StepDone := ExecuteSkill.Done;
END_ACTION

ACTION Transport1_active:
StepDone := FALSE;

//Skill auswählen
ExecuteSkill.SkillID 		:= 1320;
ExecuteSkill.SkillName	 	:= 'Name';

//Parameter setzen

ExecuteSkill.Parameter[3].ID := 3;
ExecuteSkill.Parameter[3].Name := 'Velocity';
ExecuteSkill.Parameter[3].Value := 2500;



ExecuteSkill.Parameter[4].ID := 4 ;
ExecuteSkill.Parameter[4].Name := 'Acceleration';
ExecuteSkill.Parameter[4].Value := 1000 ;



ExecuteSkill.Parameter[1].ID := 1;
ExecuteSkill.Parameter[1].Name := 'TargetPosition X';
ExecuteSkill.Parameter[1].Value := 3200 ;
ExecuteSkill.Parameter[1].StringValue := '#DP#2#XPosition' ;




ExecuteSkill.Parameter[2].ID := 2;
ExecuteSkill.Parameter[2].Name := 'TargetPosition Z';
ExecuteSkill.Parameter[2].Value := ZCookieModule;


(*
ExecuteSkill.Parameter[5].ID := ;
ExecuteSkill.Parameter[5].Name := '';
ExecuteSkill.Parameter[5].Value := ;
*)



ExecuteSkill();

StepDone := ExecuteSkill.Done;
END_ACTION

ACTION BlockBeiTopping_active:
StepDone := FALSE;

//Skill auswählen
ExecuteSkill.SkillID 		:= 1315;
ExecuteSkill.SkillName	 	:= 'Block';

//Parameter setzen

ExecuteSkill.Parameter[1].ID := 1;
ExecuteSkill.Parameter[1].Name := 'TaskID';
ExecuteSkill.Parameter[1].Value := 130;


(*
ExecuteSkill.Parameter[2].ID := ;
ExecuteSkill.Parameter[2].Name := '';
ExecuteSkill.Parameter[2].Value := ;
*)

(*
ExecuteSkill.Parameter[3].ID := ;
ExecuteSkill.Parameter[3].Name := '';
ExecuteSkill.Parameter[3].Value := ;
*)

(*
ExecuteSkill.Parameter[4].ID := ;
ExecuteSkill.Parameter[4].Name := '';
ExecuteSkill.Parameter[4].Value := ;
*)

(*
ExecuteSkill.Parameter[5].ID := ;
ExecuteSkill.Parameter[5].Name := '';
ExecuteSkill.Parameter[5].Value := ;
*)



ExecuteSkill();

StepDone := ExecuteSkill.Done;
END_ACTION

ACTION Topping_active:
StepDone := FALSE;

//Skill auswählen
ExecuteSkill.SkillID 		:= 1210;
ExecuteSkill.SkillName	 	:= 'Topping';

//Parameter setzen
(*
ExecuteSkill.Parameter[1].ID := 1;
ExecuteSkill.Parameter[1].Name := 'TaskID';
ExecuteSkill.Parameter[1].Value := 130;
*)
(*
ExecuteSkill.Parameter[2].ID := ;
ExecuteSkill.Parameter[2].Name := '';
ExecuteSkill.Parameter[2].Value := ;
*)

(*
ExecuteSkill.Parameter[3].ID := ;
ExecuteSkill.Parameter[3].Name := '';
ExecuteSkill.Parameter[3].Value := ;
*)

(*
ExecuteSkill.Parameter[4].ID := ;
ExecuteSkill.Parameter[4].Name := '';
ExecuteSkill.Parameter[4].Value := ;
*)

(*
ExecuteSkill.Parameter[5].ID := ;
ExecuteSkill.Parameter[5].Name := '';
ExecuteSkill.Parameter[5].Value := ;
*)

ExecuteSkill();

StepDone := ExecuteSkill.Done;
END_ACTION

ACTION TransportToTopping_active:
StepDone := FALSE;

//Skill auswählen
ExecuteSkill.SkillID 		:= 1320;
ExecuteSkill.SkillName	 	:= 'Transport';

//Parameter setzen

ExecuteSkill.Parameter[3].ID := 3;
ExecuteSkill.Parameter[3].Name := 'Velocity';
ExecuteSkill.Parameter[3].Value := 1500;



ExecuteSkill.Parameter[1].ID :=  1;
ExecuteSkill.Parameter[1].Name := 'TargetPosition X';
ExecuteSkill.Parameter[1].Value := 30 ;
ExecuteSkill.Parameter[1].StringValue := '#DP#2#XPosition';



ExecuteSkill.Parameter[2].ID := 2;
ExecuteSkill.Parameter[2].Name := 'TargetPosition Z';
ExecuteSkill.Parameter[2].Value := ZCremeModule ;

ExecuteSkill();

StepDone := ExecuteSkill.Done;
END_ACTION

ACTION MODULESkill_active:
StepDone := FALSE;
RecipeDone := FALSE;
//Skill auswählen
ExecuteSkill.SkillID 		:= 1010;
ExecuteSkill.SkillName	 	:= 'Cookie ausgeben';





ExecuteSkill();

StepDone := ExecuteSkill.Done;
END_ACTION

ACTION Unblock1_active:
StepDone := FALSE;

//Skill auswählen
ExecuteSkill.SkillID 		:= 1316;
ExecuteSkill.SkillName	 	:= 'Unblock';

//Parameter setzen

ExecuteSkill.Parameter[1].ID := 1;
ExecuteSkill.Parameter[1].Name := 'TaskID';
ExecuteSkill.Parameter[1].Value := 128 ;


(*
ExecuteSkill.Parameter[2].ID := ;
ExecuteSkill.Parameter[2].Name := '';
ExecuteSkill.Parameter[2].Value := ;
*)

(*
ExecuteSkill.Parameter[3].ID := ;
ExecuteSkill.Parameter[3].Name := '';
ExecuteSkill.Parameter[3].Value := ;
*)

(*
ExecuteSkill.Parameter[4].ID := ;
ExecuteSkill.Parameter[4].Name := '';
ExecuteSkill.Parameter[4].Value := ;
*)

(*
ExecuteSkill.Parameter[5].ID := ;
ExecuteSkill.Parameter[5].Name := '';
ExecuteSkill.Parameter[5].Value := ;
*)



ExecuteSkill();

StepDone := ExecuteSkill.Done;
END_ACTION

ACTION Block1_active:
StepDone := FALSE;

//Skill auswählen
ExecuteSkill.SkillID 		:= 1315;
ExecuteSkill.SkillName	 	:= 'Block';

//Parameter setzen

ExecuteSkill.Parameter[1].ID := 1;
ExecuteSkill.Parameter[1].Name := 'TaskID';
ExecuteSkill.Parameter[1].Value := 127;


(*
ExecuteSkill.Parameter[2].ID := ;
ExecuteSkill.Parameter[2].Name := '';
ExecuteSkill.Parameter[2].Value := ;
*)

(*
ExecuteSkill.Parameter[3].ID := ;
ExecuteSkill.Parameter[3].Name := '';
ExecuteSkill.Parameter[3].Value := ;
*)

(*
ExecuteSkill.Parameter[4].ID := ;
ExecuteSkill.Parameter[4].Name := '';
ExecuteSkill.Parameter[4].Value := ;
*)

(*
ExecuteSkill.Parameter[5].ID := ;
ExecuteSkill.Parameter[5].Name := '';
ExecuteSkill.Parameter[5].Value := ;
*)



ExecuteSkill();

StepDone := ExecuteSkill.Done;
END_ACTION

ACTION Transport_active:
StepDone := FALSE;

//Skill auswählen
ExecuteSkill.SkillID 		:= 1320;
ExecuteSkill.SkillName	 	:= 'Transport';

//Parameter setzen

ExecuteSkill.Parameter[3].ID :=3 ;
ExecuteSkill.Parameter[3].Name := 'Velocity';
ExecuteSkill.Parameter[3].Value := 1500;



ExecuteSkill.Parameter[1].ID :=1 ;
ExecuteSkill.Parameter[1].Name := 'TargetPosition X';
ExecuteSkill.Parameter[1].StringValue := '#DP#2#XPosition';
ExecuteSkill.Parameter[1].Value := 200 ;


ExecuteSkill.Parameter[2].ID := 2 ;
ExecuteSkill.Parameter[2].Name := 'TargetPosition Z';
ExecuteSkill.Parameter[2].Value := 90 ;



ExecuteSkill.Parameter[4].ID := 4 ;
ExecuteSkill.Parameter[4].Name := 'Acceleration';
ExecuteSkill.Parameter[4].Value := 4500;


(*
ExecuteSkill.Parameter[5].ID := ;
ExecuteSkill.Parameter[5].Name := '';
ExecuteSkill.Parameter[5].Value := ;
*)



ExecuteSkill();

StepDone := ExecuteSkill.Done;
END_ACTION

ACTION Block2_active:
StepDone := FALSE;

//Skill auswählen
ExecuteSkill.SkillID 		:= 1315;
ExecuteSkill.SkillName	 	:= 'Block';

//Parameter setzen

ExecuteSkill.Parameter[1].ID := 1;
ExecuteSkill.Parameter[1].Name := 'TaskID';
ExecuteSkill.Parameter[1].Value := 130;


(*
ExecuteSkill.Parameter[2].ID := ;
ExecuteSkill.Parameter[2].Name := '';
ExecuteSkill.Parameter[2].Value := ;
*)

(*
ExecuteSkill.Parameter[3].ID := ;
ExecuteSkill.Parameter[3].Name := '';
ExecuteSkill.Parameter[3].Value := ;
*)

(*
ExecuteSkill.Parameter[4].ID := ;
ExecuteSkill.Parameter[4].Name := '';
ExecuteSkill.Parameter[4].Value := ;
*)

(*
ExecuteSkill.Parameter[5].ID := ;
ExecuteSkill.Parameter[5].Name := '';
ExecuteSkill.Parameter[5].Value := ;
*)



ExecuteSkill();

StepDone := ExecuteSkill.Done;
END_ACTION

ACTION Block_active:
StepDone := FALSE;

//Skill auswählen
ExecuteSkill.SkillID 		:= 1315;
ExecuteSkill.SkillName	 	:= 'Block';

//Parameter setzen

ExecuteSkill.Parameter[1].ID := 1;
ExecuteSkill.Parameter[1].Name := 'TaskID';
ExecuteSkill.Parameter[1].Value := 124;


(*
ExecuteSkill.Parameter[2].ID := ;
ExecuteSkill.Parameter[2].Name := '';
ExecuteSkill.Parameter[2].Value := ;
*)

(*
ExecuteSkill.Parameter[3].ID := ;
ExecuteSkill.Parameter[3].Name := '';
ExecuteSkill.Parameter[3].Value := ;
*)

(*
ExecuteSkill.Parameter[4].ID := ;
ExecuteSkill.Parameter[4].Name := '';
ExecuteSkill.Parameter[4].Value := ;
*)

(*
ExecuteSkill.Parameter[5].ID := ;
ExecuteSkill.Parameter[5].Name := '';
ExecuteSkill.Parameter[5].Value := ;
*)



ExecuteSkill();

StepDone := ExecuteSkill.Done;
END_ACTION

ACTION Reserve_active:
StepDone := FALSE;
RecipeDone := FALSE;
//Skill auswählen
ExecuteSkill.SkillID 		:= 1310;
ExecuteSkill.SkillName	 	:= 'Reserve';

//Parameter setzen

ExecuteSkill.Parameter[1].ID := 1;
ExecuteSkill.Parameter[1].Name := 'TaskID';
ExecuteSkill.Parameter[1].Value := 123;


(*
ExecuteSkill.Parameter[2].ID := ;
ExecuteSkill.Parameter[2].Name := '';
ExecuteSkill.Parameter[2].Value := ;
*)

(*
ExecuteSkill.Parameter[3].ID := ;
ExecuteSkill.Parameter[3].Name := '';
ExecuteSkill.Parameter[3].Value := ;
*)

(*
ExecuteSkill.Parameter[4].ID := ;
ExecuteSkill.Parameter[4].Name := '';
ExecuteSkill.Parameter[4].Value := ;
*)

(*
ExecuteSkill.Parameter[5].ID := ;
ExecuteSkill.Parameter[5].Name := '';
ExecuteSkill.Parameter[5].Value := ;
*)



ExecuteSkill();

StepDone := ExecuteSkill.Done;
END_ACTION

ACTION Production0_active:
StepDone := FALSE;
RecipeDone := FALSE;
//Skill auswählen
ExecuteSkill.SkillID 		:= 1337;
ExecuteSkill.SkillName	 	:= 'Testmodul1';

ExecuteSkill();

StepDone := ExecuteSkill.Done;
END_ACTION

END_FUNCTION_BLOCK

// ---- POUs/Recipes/Recipe_10054_FreePassion_special.TcPOU
FUNCTION_BLOCK Recipe_10054_FreePassion_special
VAR_INPUT
	execute: BOOL;
	Order: DUT_RECIPEORDER;
END_VAR
VAR_OUTPUT
	RecipeInfo: DUT_RECIPEOFFER;
	RecipeDone: BOOL;
	InitDone: BOOL;
END_VAR
VAR
	userparametersum: LREAL;
	StepDone: BOOL;
	i: INT;
END_VAR

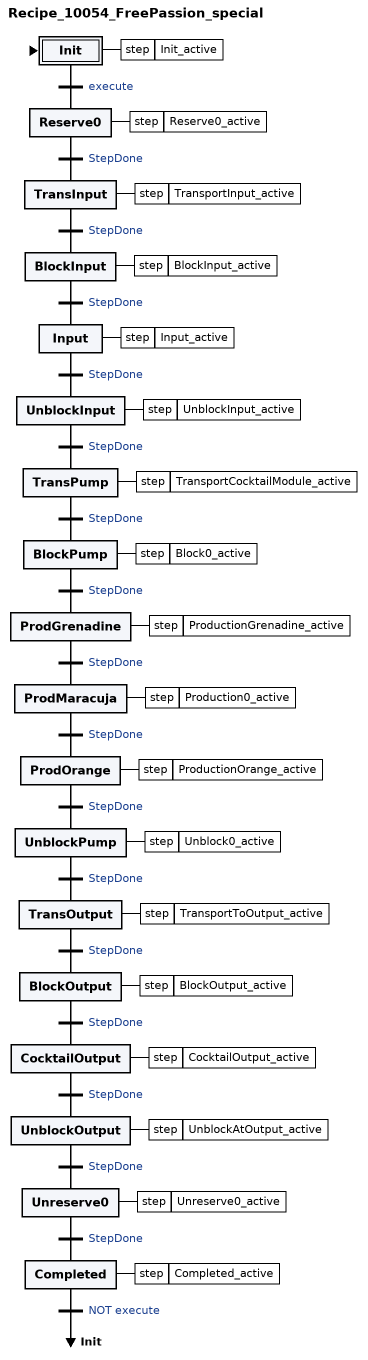
INITIAL_STEP Init:
    Init_active(N);  // step action
END_STEP
TRANSITION FROM Init TO Reserve0
    := execute;
END_TRANSITION
STEP Reserve0:
    Reserve0_active(N);  // step action
END_STEP
TRANSITION FROM Reserve0 TO TransInput
    := StepDone;
END_TRANSITION
STEP TransInput:
    TransportInput_active(N);  // step action
END_STEP
TRANSITION FROM TransInput TO BlockInput
    := StepDone;
END_TRANSITION
STEP BlockInput:
    BlockInput_active(N);  // step action
END_STEP
TRANSITION FROM BlockInput TO Input
    := StepDone;
END_TRANSITION
STEP Input:
    Input_active(N);  // step action
END_STEP
TRANSITION FROM Input TO UnblockInput
    := StepDone;
END_TRANSITION
STEP UnblockInput:
    UnblockInput_active(N);  // step action
END_STEP
TRANSITION FROM UnblockInput TO TransPump
    := StepDone;
END_TRANSITION
STEP TransPump:
    TransportCocktailModule_active(N);  // step action
END_STEP
TRANSITION FROM TransPump TO BlockPump
    := StepDone;
END_TRANSITION
STEP BlockPump:
    Block0_active(N);  // step action
END_STEP
TRANSITION FROM BlockPump TO ProdGrenadine
    := StepDone;
END_TRANSITION
STEP ProdGrenadine:
    ProductionGrenadine_active(N);  // step action
END_STEP
TRANSITION FROM ProdGrenadine TO ProdMaracuja
    := StepDone;
END_TRANSITION
STEP ProdMaracuja:
    Production0_active(N);  // step action
END_STEP
TRANSITION FROM ProdMaracuja TO ProdOrange
    := StepDone;
END_TRANSITION
STEP ProdOrange:
    ProductionOrange_active(N);  // step action
END_STEP
TRANSITION FROM ProdOrange TO UnblockPump
    := StepDone;
END_TRANSITION
STEP UnblockPump:
    Unblock0_active(N);  // step action
END_STEP
TRANSITION FROM UnblockPump TO TransOutput
    := StepDone;
END_TRANSITION
STEP TransOutput:
    TransportToOutput_active(N);  // step action
END_STEP
TRANSITION FROM TransOutput TO BlockOutput
    := StepDone;
END_TRANSITION
STEP BlockOutput:
    BlockOutput_active(N);  // step action
END_STEP
TRANSITION FROM BlockOutput TO CocktailOutput
    := StepDone;
END_TRANSITION
STEP CocktailOutput:
    CocktailOutput_active(N);  // step action
END_STEP
TRANSITION FROM CocktailOutput TO UnblockOutput
    := StepDone;
END_TRANSITION
STEP UnblockOutput:
    UnblockAtOutput_active(N);  // step action
END_STEP
TRANSITION FROM UnblockOutput TO Unreserve0
    := StepDone;
END_TRANSITION
STEP Unreserve0:
    Unreserve0_active(N);  // step action
END_STEP
TRANSITION FROM Unreserve0 TO Completed
    := StepDone;
END_TRANSITION
STEP Completed:
    Completed_active(N);  // step action
END_STEP
TRANSITION FROM Completed TO Init
    := NOT execute;
END_TRANSITION

ACTION Production0_active:
StepDone := FALSE;

userparametersum := 0;
FOR i := 1 TO UserParameterCnt DO
	IF NOT (order.UserParameter[i].Value = 0) THEN
		userparametersum := userparametersum + order.UserParameter[i].Value;
	
	END_IF
END_FOR
IF userparametersum = 0 THEN
userparametersum := -1;
END_IF
//Skill auswählen
ExecuteSkill.SkillID 		:= 1113;
ExecuteSkill.SkillName	 	:= 'Marajuca Juice';

//Parameter setzen

ExecuteSkill.Parameter[0].ID := 1;
ExecuteSkill.Parameter[0].Name := 'Quantity';
//order.userParameter[0] = amount
ExecuteSkill.Parameter[0].Value := order.UserParameter[0].Value * order.UserParameter[1].Value / userparametersum;//Summe aller Zutatenmengen;


(*
ExecuteSkill.Parameter[2].ID := ;
ExecuteSkill.Parameter[2].Name := '';
ExecuteSkill.Parameter[2].Value := ;
*)

(*
ExecuteSkill.Parameter[3].ID := ;
ExecuteSkill.Parameter[3].Name := '';
ExecuteSkill.Parameter[3].Value := ;
*)

(*
ExecuteSkill.Parameter[4].ID := ;
ExecuteSkill.Parameter[4].Name := '';
ExecuteSkill.Parameter[4].Value := ;
*)

(*
ExecuteSkill.Parameter[5].ID := ;
ExecuteSkill.Parameter[5].Name := '';
ExecuteSkill.Parameter[5].Value := ;
*)



ExecuteSkill();

StepDone := ExecuteSkill.Done;
END_ACTION

ACTION TransportInput_active:
StepDone := FALSE;

//Skill auswählen
ExecuteSkill.SkillID 		:= 1320;
ExecuteSkill.SkillName	 	:= 'Transport';

//Parameter setzen

ExecuteSkill.Parameter[3].ID := 3;
ExecuteSkill.Parameter[3].Name := 'Velocity';
ExecuteSkill.Parameter[3].Value := 1500;



ExecuteSkill.Parameter[1].ID :=  1;
ExecuteSkill.Parameter[1].Name := 'TargetPosition X';
ExecuteSkill.Parameter[1].Value := 30 ;
ExecuteSkill.Parameter[1].StringValue := '#DP#2#XPosition';



ExecuteSkill.Parameter[2].ID := 2;
ExecuteSkill.Parameter[2].Name := 'TargetPosition Z';
ExecuteSkill.Parameter[2].Value := 100;// ZCookieModule - ZCookieModuleCalibration - 2* Cookiethickness + toppingthickness+ Preasureheight  ;



(*
ExecuteSkill.Parameter[4].ID := 4;
ExecuteSkill.Parameter[4].Name := 'Acceleration';
ExecuteSkill.Parameter[4].Value := 0 ;
*)

(*
ExecuteSkill.Parameter[5].ID := ;
ExecuteSkill.Parameter[5].Name := '';
ExecuteSkill.Parameter[5].Value := ;
*)



ExecuteSkill();

StepDone := ExecuteSkill.Done;
END_ACTION

ACTION BlockOutput_active:
StepDone := FALSE;

//Skill auswählen
ExecuteSkill.SkillID 		:= 1315;
ExecuteSkill.SkillName	 	:= 'Block';

//Parameter setzen

ExecuteSkill.Parameter[1].ID := 1;
ExecuteSkill.Parameter[1].Name := 'TaskID';
ExecuteSkill.Parameter[1].Value := Order.TaskID;


(*
ExecuteSkill.Parameter[2].ID := ;
ExecuteSkill.Parameter[2].Name := '';
ExecuteSkill.Parameter[2].Value := ;
*)

(*
ExecuteSkill.Parameter[3].ID := ;
ExecuteSkill.Parameter[3].Name := '';
ExecuteSkill.Parameter[3].Value := ;
*)

(*
ExecuteSkill.Parameter[4].ID := ;
ExecuteSkill.Parameter[4].Name := '';
ExecuteSkill.Parameter[4].Value := ;
*)

(*
ExecuteSkill.Parameter[5].ID := ;
ExecuteSkill.Parameter[5].Name := '';
ExecuteSkill.Parameter[5].Value := ;
*)



ExecuteSkill();

StepDone := ExecuteSkill.Done;
END_ACTION

ACTION ProductionGrenadine_active:
StepDone := FALSE;

//Skill auswählen
ExecuteSkill.SkillID 		:= 1121;
ExecuteSkill.SkillName	 	:= 'Batida de Coco';

//Parameter setzen

ExecuteSkill.Parameter[0].ID := 1;
ExecuteSkill.Parameter[0].Name := 'Quantity';
//order.userParameter[0] = amount
ExecuteSkill.Parameter[0].Value := order.UserParameter[0].Value * order.UserParameter[3].Value / userparametersum; //Summe aller Zutatenmengen;



(*
ExecuteSkill.Parameter[2].ID := ;
ExecuteSkill.Parameter[2].Name := '';
ExecuteSkill.Parameter[2].Value := ;
*)

(*
ExecuteSkill.Parameter[3].ID := ;
ExecuteSkill.Parameter[3].Name := '';
ExecuteSkill.Parameter[3].Value := ;
*)

(*
ExecuteSkill.Parameter[4].ID := ;
ExecuteSkill.Parameter[4].Name := '';
ExecuteSkill.Parameter[4].Value := ;
*)

(*
ExecuteSkill.Parameter[5].ID := ;
ExecuteSkill.Parameter[5].Name := '';
ExecuteSkill.Parameter[5].Value := ;
*)



ExecuteSkill();

StepDone := ExecuteSkill.Done;
END_ACTION

ACTION Unreserve0_active:
StepDone := FALSE;

//Skill auswählen
ExecuteSkill.SkillID 		:= 1311;
ExecuteSkill.SkillName	 	:= 'Unreserve';

//Parameter setzen

ExecuteSkill.Parameter[1].ID := 1;
ExecuteSkill.Parameter[1].Name := 'TaskID';
ExecuteSkill.Parameter[1].Value := Order.TaskID;


(*
ExecuteSkill.Parameter[2].ID := ;
ExecuteSkill.Parameter[2].Name := '';
ExecuteSkill.Parameter[2].Val ue := ;
*)

(*
ExecuteSkill.Parameter[3].ID := ;
ExecuteSkill.Parameter[3].Name := '';
ExecuteSkill.Parameter[3].Value := ;
*)

(*
ExecuteSkill.Parameter[4].ID := ;
ExecuteSkill.Parameter[4].Name := '';
ExecuteSkill.Parameter[4].Value := ;
*)

(*
ExecuteSkill.Parameter[5].ID := ;
ExecuteSkill.Parameter[5].Name := '';
ExecuteSkill.Parameter[5].Value := ;
*)



ExecuteSkill();

StepDone := ExecuteSkill.Done;
END_ACTION

ACTION Input_active:
StepDone := FALSE;

//Skill auswählen
ExecuteSkill.SkillID 		:= 1402;
ExecuteSkill.SkillName	 	:= 'Input';

//Parameter setzen

ExecuteSkill.Parameter[1].ID := 1;
ExecuteSkill.Parameter[1].Name := 'TaskID';
ExecuteSkill.Parameter[1].Value := Order.TaskID;


(*
ExecuteSkill.Parameter[2].ID := ;
ExecuteSkill.Parameter[2].Name := '';
ExecuteSkill.Parameter[2].Value := ;
*)

(*
ExecuteSkill.Parameter[3].ID := ;
ExecuteSkill.Parameter[3].Name := '';
ExecuteSkill.Parameter[3].Value := ;
*)

(*
ExecuteSkill.Parameter[4].ID := ;
ExecuteSkill.Parameter[4].Name := '';
ExecuteSkill.Parameter[4].Value := ;
*)

(*
ExecuteSkill.Parameter[5].ID := ;
ExecuteSkill.Parameter[5].Name := '';
ExecuteSkill.Parameter[5].Value := ;
*)



ExecuteSkill();

StepDone := ExecuteSkill.Done;
END_ACTION

ACTION TransportToOutput_active:
StepDone := FALSE;

//Skill auswählen
ExecuteSkill.SkillID 		:= 1320;
ExecuteSkill.SkillName	 	:= 'Transport';

//Parameter setzen

ExecuteSkill.Parameter[3].ID := 3;
ExecuteSkill.Parameter[3].Name := 'Velocity';
ExecuteSkill.Parameter[3].Value := 280;



ExecuteSkill.Parameter[1].ID :=  1;
ExecuteSkill.Parameter[1].Name := 'TargetPosition X';
ExecuteSkill.Parameter[1].Value := 30 ;
ExecuteSkill.Parameter[1].StringValue := '#DP#2#XPosition';



ExecuteSkill.Parameter[2].ID := 2;
ExecuteSkill.Parameter[2].Name := 'TargetPosition Z';
ExecuteSkill.Parameter[2].Value := ZInputOutput;// ZCookieModule - ZCookieModuleCalibration - 2* Cookiethickness + toppingthickness+ Preasureheight  ;



(* ExecuteSkill.Parameter[4].ID := 4;
ExecuteSkill.Parameter[4].Name := 'Acceleration';
ExecuteSkill.Parameter[4].Value :=0 ;

*)
(*
ExecuteSkill.Parameter[5].ID := ;
ExecuteSkill.Parameter[5].Name := '';
ExecuteSkill.Parameter[5].Value := ;
*)



ExecuteSkill();

StepDone := ExecuteSkill.Done;
END_ACTION

ACTION ProductionOrange_active:
StepDone := FALSE;

//Skill auswählen
ExecuteSkill.SkillID 		:= 1117;
ExecuteSkill.SkillName	 	:= 'Orange';

//Parameter setzen

ExecuteSkill.Parameter[0].ID := 1;
ExecuteSkill.Parameter[0].Name := 'Quantity';
//order.userParameter[0] = amount
ExecuteSkill.Parameter[0].Value := order.UserParameter[0].Value * order.UserParameter[2].Value / userparametersum;//Summe aller Zutatenmengen;



(*
ExecuteSkill.Parameter[2].ID := ;
ExecuteSkill.Parameter[2].Name := '';
ExecuteSkill.Parameter[2].Value := ;
*)

(*
ExecuteSkill.Parameter[3].ID := ;
ExecuteSkill.Parameter[3].Name := '';
ExecuteSkill.Parameter[3].Value := ;
*)

(*
ExecuteSkill.Parameter[4].ID := ;
ExecuteSkill.Parameter[4].Name := '';
ExecuteSkill.Parameter[4].Value := ;
*)

(*
ExecuteSkill.Parameter[5].ID := ;
ExecuteSkill.Parameter[5].Name := '';
ExecuteSkill.Parameter[5].Value := ;
*)



ExecuteSkill();

StepDone := ExecuteSkill.Done;
END_ACTION

ACTION UnblockAtOutput_active:
StepDone := FALSE;

//Skill auswählen
ExecuteSkill.SkillID 		:= 1316;
ExecuteSkill.SkillName	 	:= 'Unblock';

//Parameter setzen

ExecuteSkill.Parameter[1].ID := 1;
ExecuteSkill.Parameter[1].Name := 'TaskID';
ExecuteSkill.Parameter[1].Value := Order.TaskID;


(*
ExecuteSkill.Parameter[2].ID := ;
ExecuteSkill.Parameter[2].Name := '';
ExecuteSkill.Parameter[2].Value := ;
*)

(*
ExecuteSkill.Parameter[3].ID := ;
ExecuteSkill.Parameter[3].Name := '';
ExecuteSkill.Parameter[3].Value := ;
*)

(*
ExecuteSkill.Parameter[4].ID := ;
ExecuteSkill.Parameter[4].Name := '';
ExecuteSkill.Parameter[4].Value := ;
*)

(*
ExecuteSkill.Parameter[5].ID := ;
ExecuteSkill.Parameter[5].Name := '';
ExecuteSkill.Parameter[5].Value := ;
*)



ExecuteSkill();

StepDone := ExecuteSkill.Done;
END_ACTION

ACTION CocktailOutput_active:
StepDone := FALSE;

//Skill auswählen
ExecuteSkill.SkillID 		:= 1403;
ExecuteSkill.SkillName	 	:= 'Output';

//Parameter setzen

ExecuteSkill.Parameter[1].ID := 1;
ExecuteSkill.Parameter[1].Name := 'TaskID';
ExecuteSkill.Parameter[1].Value := Order.TaskID;


(*
ExecuteSkill.Parameter[2].ID := ;
ExecuteSkill.Parameter[2].Name := '';
ExecuteSkill.Parameter[2].Value := ;
*)

(*
ExecuteSkill.Parameter[3].ID := ;
ExecuteSkill.Parameter[3].Name := '';
ExecuteSkill.Parameter[3].Value := ;
*)

(*
ExecuteSkill.Parameter[4].ID := ;
ExecuteSkill.Parameter[4].Name := '';
ExecuteSkill.Parameter[4].Value := ;
*)

(*
ExecuteSkill.Parameter[5].ID := ;
ExecuteSkill.Parameter[5].Name := '';
ExecuteSkill.Parameter[5].Value := ;
*)

ExecuteSkill();

StepDone := ExecuteSkill.Done;
END_ACTION

ACTION Completed_active:
RecipeDone := TRUE;
StepDone := FALSE;
END_ACTION

ACTION UnblockInput_active:
StepDone := FALSE;

//Skill auswählen
ExecuteSkill.SkillID 		:= 1316;
ExecuteSkill.SkillName	 	:= 'Unblock';

//Parameter setzen

ExecuteSkill.Parameter[1].ID := 1;
ExecuteSkill.Parameter[1].Name := 'TaskID';
ExecuteSkill.Parameter[1].Value := Order.TaskID;


(*
ExecuteSkill.Parameter[2].ID := ;
ExecuteSkill.Parameter[2].Name := '';
ExecuteSkill.Parameter[2].Value := ;
*)

(*
ExecuteSkill.Parameter[3].ID := ;
ExecuteSkill.Parameter[3].Name := '';
ExecuteSkill.Parameter[3].Value := ;
*)

(*
ExecuteSkill.Parameter[4].ID := ;
ExecuteSkill.Parameter[4].Name := '';
ExecuteSkill.Parameter[4].Value := ;
*)

(*
ExecuteSkill.Parameter[5].ID := ;
ExecuteSkill.Parameter[5].Name := '';
ExecuteSkill.Parameter[5].Value := ;
*)



ExecuteSkill();

StepDone := ExecuteSkill.Done;
END_ACTION

ACTION Unblock0_active:
StepDone := FALSE;

//Skill auswählen
ExecuteSkill.SkillID 		:= 1316;
ExecuteSkill.SkillName	 	:= 'Unblock';

//Parameter setzen

ExecuteSkill.Parameter[1].ID := 1;
ExecuteSkill.Parameter[1].Name := 'TaskID';
ExecuteSkill.Parameter[1].Value := Order.TaskID;


(*
ExecuteSkill.Parameter[2].ID := ;
ExecuteSkill.Parameter[2].Name := '';
ExecuteSkill.Parameter[2].Value := ;
*)

(*
ExecuteSkill.Parameter[3].ID := ;
ExecuteSkill.Parameter[3].Name := '';
ExecuteSkill.Parameter[3].Value := ;
*)

(*
ExecuteSkill.Parameter[4].ID := ;
ExecuteSkill.Parameter[4].Name := '';
ExecuteSkill.Parameter[4].Value := ;
*)

(*
ExecuteSkill.Parameter[5].ID := ;
ExecuteSkill.Parameter[5].Name := '';
ExecuteSkill.Parameter[5].Value := ;
*)



ExecuteSkill();

StepDone := ExecuteSkill.Done;
END_ACTION

ACTION TransportCocktailModule_active:
StepDone := FALSE;

//Skill auswählen
ExecuteSkill.SkillID 		:= 1320;
ExecuteSkill.SkillName	 	:= 'Transport';

//Parameter setzen

ExecuteSkill.Parameter[3].ID := 3;
ExecuteSkill.Parameter[3].Name := 'Velocity';
ExecuteSkill.Parameter[3].Value := 1000;



ExecuteSkill.Parameter[1].ID :=  1;
ExecuteSkill.Parameter[1].Name := 'TargetPosition X';
ExecuteSkill.Parameter[1].Value := 30 ;
ExecuteSkill.Parameter[1].StringValue := '#DP#2#XPosition';



ExecuteSkill.Parameter[2].ID := 2;
ExecuteSkill.Parameter[2].Name := 'TargetPosition Z';
ExecuteSkill.Parameter[2].Value := 40;// ZCookieModule - ZCookieModuleCalibration - 2* Cookiethickness + toppingthickness+ Preasureheight  ;



(*
ExecuteSkill.Parameter[4].ID := 4;
ExecuteSkill.Parameter[4].Name := 'Acceleration';
ExecuteSkill.Parameter[4].Value := 0 ;
*)

(*
ExecuteSkill.Parameter[5].ID := ;
ExecuteSkill.Parameter[5].Name := '';
ExecuteSkill.Parameter[5].Value := ;
*)



ExecuteSkill();

StepDone := ExecuteSkill.Done;
END_ACTION

ACTION Init_active:
RecipeDone := FALSE;

// Initialisation of Recipe Parameters an name etc
RecipeInfo.Name := 'Free Passion special';
RecipeInfo.Description := 'Sweet cocktail combining the sourness of maracuja and orange juice with the taste of Coco';
RecipeInfo.Dummy := FALSE;
RecipeInfo.RecipeID := 10054; 	// 
Initdone := TRUE;

FOR i := 0 TO UserParameterCnt DO
	IF Order.UserParameter[i].Value = 0 THEN
		order.UserParameter[i].Value := RecipeInfo.UserParameter[i].Default;
	END_IF
END_FOR
//Parameter 0:

	RecipeInfo.UserParameter[0].Dummy 		:= FALSE;
	RecipeInfo.UserParameter[0].Default		:= 200;
	RecipeInfo.UserParameter[0].Description	:= 'Gives the total fluid amount in the glass';
	RecipeInfo.UserParameter[0].MaxValue	:= 200;
	RecipeInfo.UserParameter[0].MinValue	:= 10;
	RecipeInfo.UserParameter[0].Name		:= 'Total Liquid Amount';
	RecipeInfo.UserParameter[0].Unit		:= 'ml';
	
//Parameter 1:

	RecipeInfo.UserParameter[1].Dummy 		:= FALSE;
	RecipeInfo.UserParameter[1].Default		:= 50;
	RecipeInfo.UserParameter[1].Description	:= 'Maracuja Juice';
	RecipeInfo.UserParameter[1].MaxValue	:= 100;
	RecipeInfo.UserParameter[1].MinValue	:= 1;
	RecipeInfo.UserParameter[1].Name		:= 'Maracuja Juice';
	RecipeInfo.UserParameter[1].Unit		:= 'ml';
	
//Parameter 2:

	RecipeInfo.UserParameter[2].Dummy 		:= FALSE;
	RecipeInfo.UserParameter[2].Default		:= 35;
	RecipeInfo.UserParameter[2].Description	:= 'Orange Juice';
	RecipeInfo.UserParameter[2].MaxValue	:= 100;
	RecipeInfo.UserParameter[2].MinValue	:= 1;
	RecipeInfo.UserParameter[2].Name		:= 'Orange Juice';
	RecipeInfo.UserParameter[2].Unit		:= 'ml';

//Parameter 3:

	RecipeInfo.UserParameter[3].Dummy 		:= FALSE;
	RecipeInfo.UserParameter[3].Default		:= 15;
	RecipeInfo.UserParameter[3].Description	:= 'Batida de Coco';
	RecipeInfo.UserParameter[3].MaxValue	:= 50;
	RecipeInfo.UserParameter[3].MinValue	:= 1;
	RecipeInfo.UserParameter[3].Name		:= 'Batida de Coco';
	RecipeInfo.UserParameter[3].Unit		:= 'ml';
	
	
	
//Parameter 1:
(*
	RecipeInfo.UserParameter[1].Dummy 		:= 
	RecipeInfo.UserParameter[1].Default		:=
	RecipeInfo.UserParameter[1].Description	:=
	RecipeInfo.UserParameter[1].MaxValue	:=
	RecipeInfo.UserParameter[1].MinValue	:=
	RecipeInfo.UserParameter[1].Name		:=
	RecipeInfo.UserParameter[1].Unit		:=
*)
//Parameter 2:

(*
	RecipeInfo.UserParameter[2].Dummy 		:= 
	RecipeInfo.UserParameter[2].Default		:=
	RecipeInfo.UserParameter[2].Description	:=
	RecipeInfo.UserParameter[2].MaxValue	:=
	RecipeInfo.UserParameter[2].MinValue	:=
	RecipeInfo.UserParameter[2].Name		:=
	RecipeInfo.UserParameter[2].Unit		:=
*)

//Parameter 3:

(*
	RecipeInfo.UserParameter[3].Dummy 		:= 
	RecipeInfo.UserParameter[3].Default		:=
	RecipeInfo.UserParameter[3].Description	:=
	RecipeInfo.UserParameter[3].MaxValue	:=
	RecipeInfo.UserParameter[3].MinValue	:=
	RecipeInfo.UserParameter[3].Name		:=
	RecipeInfo.UserParameter[3].Unit		:=
*)

//Parameter 4:

(*
	RecipeInfo.UserParameter[4].Dummy 		:= 
	RecipeInfo.UserParameter[4].Default		:=
	RecipeInfo.UserParameter[4].Description	:=
	RecipeInfo.UserParameter[4].MaxValue	:=
	RecipeInfo.UserParameter[4].MinValue	:=
	RecipeInfo.UserParameter[4].Name		:=
	RecipeInfo.UserParameter[4].Unit		:=
*)


//Parameter 5:

(*
	RecipeInfo.UserParameter[5].Dummy 		:= 
	RecipeInfo.UserParameter[5].Default		:=
	RecipeInfo.UserParameter[5].Description	:=
	RecipeInfo.UserParameter[5].MaxValue	:=
	RecipeInfo.UserParameter[5].MinValue	:=
	RecipeInfo.UserParameter[5].Name		:=
	RecipeInfo.UserParameter[5].Unit		:=
*)
END_ACTION

ACTION Block0_active:
StepDone := FALSE;

//Skill auswählen
ExecuteSkill.SkillID 		:= 1315;
ExecuteSkill.SkillName	 	:= 'Block';

//Parameter setzen

ExecuteSkill.Parameter[1].ID := 1;
ExecuteSkill.Parameter[1].Name := 'TaskID';
ExecuteSkill.Parameter[1].Value := Order.TaskID;


(*
ExecuteSkill.Parameter[2].ID := ;
ExecuteSkill.Parameter[2].Name := '';
ExecuteSkill.Parameter[2].Value := ;
*)

(*
ExecuteSkill.Parameter[3].ID := ;
ExecuteSkill.Parameter[3].Name := '';
ExecuteSkill.Parameter[3].Value := ;
*)

(*
ExecuteSkill.Parameter[4].ID := ;
ExecuteSkill.Parameter[4].Name := '';
ExecuteSkill.Parameter[4].Value := ;
*)

(*
ExecuteSkill.Parameter[5].ID := ;
ExecuteSkill.Parameter[5].Name := '';
ExecuteSkill.Parameter[5].Value := ;
*)



ExecuteSkill();

StepDone := ExecuteSkill.Done;
END_ACTION

ACTION Reserve0_active:
StepDone := FALSE;
RecipeDone := FALSE;
//Skill auswählen
ExecuteSkill.SkillID 		:= 1310;
ExecuteSkill.SkillName	 	:= 'Reserve';

//Parameter setzen

ExecuteSkill.Parameter[1].ID := 1;
ExecuteSkill.Parameter[1].Name := 'TaskID';
ExecuteSkill.Parameter[1].Value := Order.TaskID;


(*
ExecuteSkill.Parameter[2].ID := ;
ExecuteSkill.Parameter[2].Name := '';
ExecuteSkill.Parameter[2].Value := ;
*)

(*
ExecuteSkill.Parameter[3].ID := ;
ExecuteSkill.Parameter[3].Name := '';
ExecuteSkill.Parameter[3].Value := ;
*)

(*
ExecuteSkill.Parameter[4].ID := ;
ExecuteSkill.Parameter[4].Name := '';
ExecuteSkill.Parameter[4].Value := ;
*)

(*
ExecuteSkill.Parameter[5].ID := ;
ExecuteSkill.Parameter[5].Name := '';
ExecuteSkill.Parameter[5].Value := ;
*)



ExecuteSkill();

StepDone := ExecuteSkill.Done;
END_ACTION

ACTION BlockInput_active:
StepDone := FALSE;

//Skill auswählen
ExecuteSkill.SkillID 		:= 1315;
ExecuteSkill.SkillName	 	:= 'Block';

//Parameter setzen

ExecuteSkill.Parameter[1].ID := 1;
ExecuteSkill.Parameter[1].Name := 'TaskID';
ExecuteSkill.Parameter[1].Value := Order.TaskID;


(*
ExecuteSkill.Parameter[2].ID := ;
ExecuteSkill.Parameter[2].Name := '';
ExecuteSkill.Parameter[2].Value := ;
*)

(*
ExecuteSkill.Parameter[3].ID := ;
ExecuteSkill.Parameter[3].Name := '';
ExecuteSkill.Parameter[3].Value := ;
*)

(*
ExecuteSkill.Parameter[4].ID := ;
ExecuteSkill.Parameter[4].Name := '';
ExecuteSkill.Parameter[4].Value := ;
*)

(*
ExecuteSkill.Parameter[5].ID := ;
ExecuteSkill.Parameter[5].Name := '';
ExecuteSkill.Parameter[5].Value := ;
*)



ExecuteSkill();

StepDone := ExecuteSkill.Done;
END_ACTION

END_FUNCTION_BLOCK

// ---- POUs/Recipes/Recipe_10052_Orangenschorle.TcPOU
FUNCTION_BLOCK Recipe_10052_Orangenschorle
VAR_INPUT
	execute: BOOL;
	Order: DUT_RECIPEORDER;
END_VAR
VAR_OUTPUT
	RecipeInfo: DUT_RECIPEOFFER;
	RecipeDone: BOOL;
	InitDone: BOOL;
	Ready: BOOL;
END_VAR
VAR
	userparametersum: LREAL;
	StepDone: BOOL;
	i: INT;
	Command: ARRAY[1..5] OF DUT_RecipeCommand;
	NextSkill: BOOL;
	SectionReady: BOOL;
END_VAR

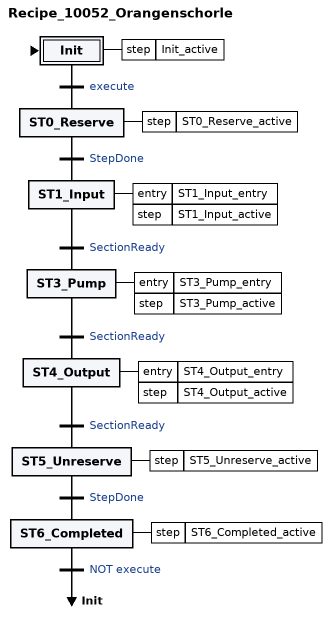
INITIAL_STEP Init:
    Init_active(N);  // step action
END_STEP
TRANSITION FROM Init TO ST0_Reserve
    := execute;
END_TRANSITION
STEP ST0_Reserve:
    ST0_Reserve_active(N);  // step action
END_STEP
TRANSITION FROM ST0_Reserve TO ST1_Input
    := StepDone;
END_TRANSITION
STEP ST1_Input:
    ST1_Input_entry(P1);  // entry action
    ST1_Input_active(N);  // step action
END_STEP
TRANSITION FROM ST1_Input TO ST3_Pump
    := SectionReady;
END_TRANSITION
STEP ST3_Pump:
    ST3_Pump_entry(P1);  // entry action
    ST3_Pump_active(N);  // step action
END_STEP
TRANSITION FROM ST3_Pump TO ST4_Output
    := SectionReady;
END_TRANSITION
STEP ST4_Output:
    ST4_Output_entry(P1);  // entry action
    ST4_Output_active(N);  // step action
END_STEP
TRANSITION FROM ST4_Output TO ST5_Unreserve
    := SectionReady;
END_TRANSITION
STEP ST5_Unreserve:
    ST5_Unreserve_active(N);  // step action
END_STEP
TRANSITION FROM ST5_Unreserve TO ST6_Completed
    := StepDone;
END_TRANSITION
STEP ST6_Completed:
    ST6_Completed_active(N);  // step action
END_STEP
TRANSITION FROM ST6_Completed TO Init
    := NOT execute;
END_TRANSITION

ACTION ST13_UnblockInput_active:
//RT: 2014.11.23: Gibt Mover Position Frei
StepDone := FALSE;

//Skill auswählen
ExecuteSkill.SkillID 		:= 1316;
ExecuteSkill.SkillName	 	:= 'Unblock';

//Parameter setzen

ExecuteSkill.Parameter[1].ID := 1;
ExecuteSkill.Parameter[1].Name := 'TaskID';
ExecuteSkill.Parameter[1].Value := Order.TaskID;


(*
ExecuteSkill.Parameter[2].ID := ;
ExecuteSkill.Parameter[2].Name := '';
ExecuteSkill.Parameter[2].Value := ;
*)

(*
ExecuteSkill.Parameter[3].ID := ;
ExecuteSkill.Parameter[3].Name := '';
ExecuteSkill.Parameter[3].Value := ;
*)

(*
ExecuteSkill.Parameter[4].ID := ;
ExecuteSkill.Parameter[4].Name := '';
ExecuteSkill.Parameter[4].Value := ;
*)

(*
ExecuteSkill.Parameter[5].ID := ;
ExecuteSkill.Parameter[5].Name := '';
ExecuteSkill.Parameter[5].Value := ;
*)



ExecuteSkill();

StepDone := ExecuteSkill.Done;
END_ACTION

ACTION ST43_UnblockOutput_active:
//RT: 2014.11.23: Gibt Mover Position Frei
StepDone := FALSE;

//Skill auswählen
ExecuteSkill.SkillID 		:= 1316;
ExecuteSkill.SkillName	 	:= 'Unblock';

//Parameter setzen

ExecuteSkill.Parameter[1].ID := 1;
ExecuteSkill.Parameter[1].Name := 'TaskID';
ExecuteSkill.Parameter[1].Value := Order.TaskID;


(*
ExecuteSkill.Parameter[2].ID := ;
ExecuteSkill.Parameter[2].Name := '';
ExecuteSkill.Parameter[2].Value := ;
*)

(*
ExecuteSkill.Parameter[3].ID := ;
ExecuteSkill.Parameter[3].Name := '';
ExecuteSkill.Parameter[3].Value := ;
*)

(*
ExecuteSkill.Parameter[4].ID := ;
ExecuteSkill.Parameter[4].Name := '';
ExecuteSkill.Parameter[4].Value := ;
*)

(*
ExecuteSkill.Parameter[5].ID := ;
ExecuteSkill.Parameter[5].Name := '';
ExecuteSkill.Parameter[5].Value := ;
*)



ExecuteSkill();

StepDone := ExecuteSkill.Done;
END_ACTION

ACTION ST1_Input_entry:
SectionReady := FALSE;
END_ACTION

ACTION ST3_Pump_entry:
SectionReady := FALSE;
END_ACTION

ACTION ST1_Input_active:
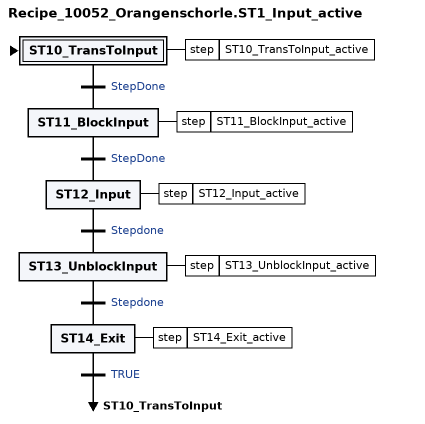
INITIAL_STEP ST10_TransToInput:
    ST10_TransToInput_active(N);  // step action
END_STEP
TRANSITION FROM ST10_TransToInput TO ST11_BlockInput
    := StepDone;
END_TRANSITION
STEP ST11_BlockInput:
    ST11_BlockInput_active(N);  // step action
END_STEP
TRANSITION FROM ST11_BlockInput TO ST12_Input
    := StepDone;
END_TRANSITION
STEP ST12_Input:
    ST12_Input_active(N);  // step action
END_STEP
TRANSITION FROM ST12_Input TO ST13_UnblockInput
    := Stepdone;
END_TRANSITION
STEP ST13_UnblockInput:
    ST13_UnblockInput_active(N);  // step action
END_STEP
TRANSITION FROM ST13_UnblockInput TO ST14_Exit
    := Stepdone;
END_TRANSITION
STEP ST14_Exit:
    ST14_Exit_active(N);  // step action
END_STEP
TRANSITION FROM ST14_Exit TO ST10_TransToInput
    := TRUE;
END_TRANSITION
END_ACTION

ACTION ST5_Unreserve_active:
//RT: 2014.11.23: Mover Freigeben
StepDone := FALSE;

//Skill auswählen
ExecuteSkill.SkillID 		:= 1311;
ExecuteSkill.SkillName	 	:= 'Unreserve';

//Parameter setzen

ExecuteSkill.Parameter[1].ID := 1;
ExecuteSkill.Parameter[1].Name := 'TaskID';
ExecuteSkill.Parameter[1].Value := Order.TaskID;


(*
ExecuteSkill.Parameter[2].ID := ;
ExecuteSkill.Parameter[2].Name := '';
ExecuteSkill.Parameter[2].Val ue := ;
*)

(*
ExecuteSkill.Parameter[3].ID := ;
ExecuteSkill.Parameter[3].Name := '';
ExecuteSkill.Parameter[3].Value := ;
*)

(*
ExecuteSkill.Parameter[4].ID := ;
ExecuteSkill.Parameter[4].Name := '';
ExecuteSkill.Parameter[4].Value := ;
*)

(*
ExecuteSkill.Parameter[5].ID := ;
ExecuteSkill.Parameter[5].Name := '';
ExecuteSkill.Parameter[5].Value := ;
*)



ExecuteSkill();

StepDone := ExecuteSkill.Done;
END_ACTION

ACTION ST1_Reserve0_active:
//RT: 2014.11.23: Reservire einen Mover

StepDone := FALSE;
RecipeDone := FALSE;
//Skill auswählen
ExecuteSkill.SkillID 		:= 1310;
ExecuteSkill.SkillName	 	:= 'Reserve';

//Parameter setzen

ExecuteSkill.Parameter[1].ID := 1;
ExecuteSkill.Parameter[1].Name := 'TaskID';
ExecuteSkill.Parameter[1].Value := Order.TaskID;

(*
ExecuteSkill.Parameter[2].ID := ;
ExecuteSkill.Parameter[2].Name := '';
ExecuteSkill.Parameter[2].Value := ;
*)

(*
ExecuteSkill.Parameter[3].ID := ;
ExecuteSkill.Parameter[3].Name := '';
ExecuteSkill.Parameter[3].Value := ;
*)

(*
ExecuteSkill.Parameter[4].ID := ;
ExecuteSkill.Parameter[4].Name := '';
ExecuteSkill.Parameter[4].Value := ;
*)

(*
ExecuteSkill.Parameter[5].ID := ;
ExecuteSkill.Parameter[5].Name := '';
ExecuteSkill.Parameter[5].Value := ;
*)

ExecuteSkill();

StepDone := ExecuteSkill.Done;
END_ACTION

ACTION ST32b_Dose_active:
//RT: 2014.11.23: Die Dosir Skills anlegen
StepDone := FALSE;

//Skill auswählen
ExecuteSkill.SkillID 		:= Command[i].SkillID;
ExecuteSkill.SkillName	 	:= Command[i].SkillName;
//Parameter setzen

ExecuteSkill.Parameter[0].ID := 1;
ExecuteSkill.Parameter[0].Name := 'Quantity';
//order.userParameter[0] = amount
ExecuteSkill.Parameter[0].Value := order.UserParameter[0].Value * order.UserParameter[i].Value / userparametersum ;//Summe aller Zutatenmengen;

(*
ExecuteSkill.Parameter[2].ID := ;
ExecuteSkill.Parameter[2].Name := '';
ExecuteSkill.Parameter[2].Value := ;
*)

(*
ExecuteSkill.Parameter[3].ID := ;
ExecuteSkill.Parameter[3].Name := '';
ExecuteSkill.Parameter[3].Value := ;
*)

(*
ExecuteSkill.Parameter[4].ID := ;
ExecuteSkill.Parameter[4].Name := '';
ExecuteSkill.Parameter[4].Value := ;
*)

(*
ExecuteSkill.Parameter[5].ID := ;
ExecuteSkill.Parameter[5].Name := '';
ExecuteSkill.Parameter[5].Value := ;
*)


ExecuteSkill();

StepDone := ExecuteSkill.Done;

i := i + 1 ;

IF i = 6 THEN
	NextSkill := FALSE;
ELSIF Command[i].SkillID = 0 THEN
	NextSkill := FALSE;
ELSE
	NextSkill := TRUE;
END_IF
END_ACTION

ACTION ST11_BlockInput_active:
//RT: 2014.11.23: Blockirt den Mover an Position
StepDone := FALSE;

//Skill auswählen
ExecuteSkill.SkillID 		:= 1315;
ExecuteSkill.SkillName	 	:= 'Block';

//Parameter setzen

ExecuteSkill.Parameter[1].ID := 1;
ExecuteSkill.Parameter[1].Name := 'TaskID';
ExecuteSkill.Parameter[1].Value := Order.TaskID;


(*
ExecuteSkill.Parameter[2].ID := ;
ExecuteSkill.Parameter[2].Name := '';
ExecuteSkill.Parameter[2].Value := ;
*)

(*
ExecuteSkill.Parameter[3].ID := ;
ExecuteSkill.Parameter[3].Name := '';
ExecuteSkill.Parameter[3].Value := ;
*)

(*
ExecuteSkill.Parameter[4].ID := ;
ExecuteSkill.Parameter[4].Name := '';
ExecuteSkill.Parameter[4].Value := ;
*)

(*
ExecuteSkill.Parameter[5].ID := ;
ExecuteSkill.Parameter[5].Name := '';
ExecuteSkill.Parameter[5].Value := ;
*)



ExecuteSkill();

StepDone := ExecuteSkill.Done;
END_ACTION

ACTION Init_active:
//RT: 2014.11.23: Vorbereiten der daten und der HMI
RecipeDone := FALSE;

// Initialisation of Recipe Parameters an name etc
RecipeInfo.Name := 'Orange Spritzer';
RecipeInfo.Description := 'Simple, but refreshing combination of orange and water';
RecipeInfo.Dummy := FALSE;
RecipeInfo.RecipeID := 10052; 	// 
Initdone := TRUE;

//RT: 2014.11.23: wenn weniger als 5 alle leeren skills SkillID := 0
Command[1].SkillID := 1117;
Command[1].SkillName := 'Orange Juice';
Command[1].Quantity := 50;

Command[2].SkillID := 1121;
Command[2].SkillName := 'Water';
Command[2].Quantity := 50;

Command[3].SkillID := 0;
Command[3].SkillName := 'Nothing';
Command[3].Quantity := 0;

Command[4].SkillID := 0;
Command[4].SkillName := 'Nothing';
Command[4].Quantity := 0;

Command[5].SkillID := 0;
Command[5].SkillName := 'Nothing';
Command[5].Quantity := 0;








//Parameter 0:

	RecipeInfo.UserParameter[0].Dummy 		:= FALSE;
	RecipeInfo.UserParameter[0].Default		:= 200;
	RecipeInfo.UserParameter[0].Description	:= 'Gives the total fluid amount in the glass';
	RecipeInfo.UserParameter[0].MaxValue	:= 200;
	RecipeInfo.UserParameter[0].MinValue	:= 10;
	RecipeInfo.UserParameter[0].Name		:= 'Total Liquid Amount';
	RecipeInfo.UserParameter[0].Unit		:= 'ml';
	
//Parameter 1-5:
FOR i := 1 TO 5 DO
	IF Command[i].SkillID = 0 THEN
		RecipeInfo.UserParameter[i].Dummy 		:= TRUE;
	ELSE
		RecipeInfo.UserParameter[i].Dummy 		:= FALSE;
		RecipeInfo.UserParameter[i].Default		:= Command[i].Quantity;
		RecipeInfo.UserParameter[i].Description	:= Command[i].SkillName;
		RecipeInfo.UserParameter[i].MaxValue	:= 100;
		RecipeInfo.UserParameter[i].MinValue	:= 1;
		RecipeInfo.UserParameter[i].Name		:= Command[i].SkillName;
		RecipeInfo.UserParameter[i].Unit		:= 'ml';	
	END_IF
END_FOR
END_ACTION

ACTION ST30_TransPump_active:
//RT: 2014.11.23: Mover zum Pump
StepDone := FALSE;

//Skill auswählen
ExecuteSkill.SkillID 		:= 1320;
ExecuteSkill.SkillName	 	:= 'Transport';

//Parameter setzen

ExecuteSkill.Parameter[3].ID := 3;
ExecuteSkill.Parameter[3].Name := 'Velocity';
ExecuteSkill.Parameter[3].Value := 1000;



ExecuteSkill.Parameter[1].ID :=  1;
ExecuteSkill.Parameter[1].Name := 'TargetPosition X';
ExecuteSkill.Parameter[1].Value := 30 ;
ExecuteSkill.Parameter[1].StringValue := '#DP#2#XPosition';



ExecuteSkill.Parameter[2].ID := 2;
ExecuteSkill.Parameter[2].Name := 'TargetPosition Z';
ExecuteSkill.Parameter[2].Value := 40;// ZCookieModule - ZCookieModuleCalibration - 2* Cookiethickness + toppingthickness+ Preasureheight  ;



(*
ExecuteSkill.Parameter[4].ID := 4;
ExecuteSkill.Parameter[4].Name := 'Acceleration';
ExecuteSkill.Parameter[4].Value := 0 ;
*)

(*
ExecuteSkill.Parameter[5].ID := ;
ExecuteSkill.Parameter[5].Name := '';
ExecuteSkill.Parameter[5].Value := ;
*)



ExecuteSkill();

StepDone := ExecuteSkill.Done;
END_ACTION

ACTION ST4_Output_active:
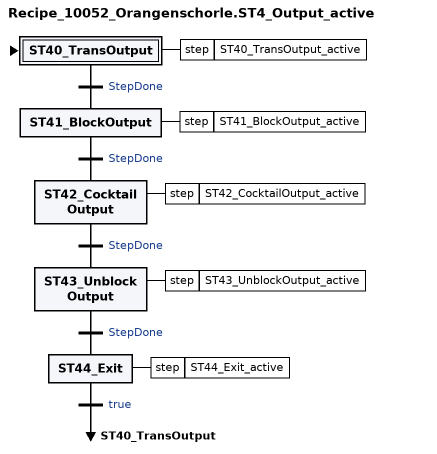
INITIAL_STEP ST40_TransOutput:
    ST40_TransOutput_active(N);  // step action
END_STEP
TRANSITION FROM ST40_TransOutput TO ST41_BlockOutput
    := StepDone;
END_TRANSITION
STEP ST41_BlockOutput:
    ST41_BlockOutput_active(N);  // step action
END_STEP
TRANSITION FROM ST41_BlockOutput TO ST42_CocktailOutput
    := StepDone;
END_TRANSITION
STEP ST42_CocktailOutput:
    ST42_CocktailOutput_active(N);  // step action
END_STEP
TRANSITION FROM ST42_CocktailOutput TO ST43_UnblockOutput
    := StepDone;
END_TRANSITION
STEP ST43_UnblockOutput:
    ST43_UnblockOutput_active(N);  // step action
END_STEP
TRANSITION FROM ST43_UnblockOutput TO ST44_Exit
    := StepDone;
END_TRANSITION
STEP ST44_Exit:
    ST44_Exit_active(N);  // step action
END_STEP
TRANSITION FROM ST44_Exit TO ST40_TransOutput
    := true;
END_TRANSITION
END_ACTION

ACTION ST0_Reserve_active:
//RT: 2014.11.23: Reservire einen Mover

StepDone := FALSE;
RecipeDone := FALSE;
//Skill auswählen
ExecuteSkill.SkillID 		:= 1310;
ExecuteSkill.SkillName	 	:= 'Reserve';

//Parameter setzen

ExecuteSkill.Parameter[1].ID := 1;
ExecuteSkill.Parameter[1].Name := 'TaskID';
ExecuteSkill.Parameter[1].Value := Order.TaskID;

(*
ExecuteSkill.Parameter[2].ID := ;
ExecuteSkill.Parameter[2].Name := '';
ExecuteSkill.Parameter[2].Value := ;
*)

(*
ExecuteSkill.Parameter[3].ID := ;
ExecuteSkill.Parameter[3].Name := '';
ExecuteSkill.Parameter[3].Value := ;
*)

(*
ExecuteSkill.Parameter[4].ID := ;
ExecuteSkill.Parameter[4].Name := '';
ExecuteSkill.Parameter[4].Value := ;
*)

(*
ExecuteSkill.Parameter[5].ID := ;
ExecuteSkill.Parameter[5].Name := '';
ExecuteSkill.Parameter[5].Value := ;
*)

ExecuteSkill();

StepDone := ExecuteSkill.Done;
END_ACTION

ACTION ST40_TransOutput_active:
//RT: 2014.11.23: Mover zum Output
StepDone := FALSE;

//Skill auswählen
ExecuteSkill.SkillID 		:= 1320;
ExecuteSkill.SkillName	 	:= 'Transport';

//Parameter setzen

ExecuteSkill.Parameter[3].ID := 3;
ExecuteSkill.Parameter[3].Name := 'Velocity';
ExecuteSkill.Parameter[3].Value := 300;



ExecuteSkill.Parameter[1].ID :=  1;
ExecuteSkill.Parameter[1].Name := 'TargetPosition X';
ExecuteSkill.Parameter[1].Value := 30 ;
ExecuteSkill.Parameter[1].StringValue := '#DP#2#XPosition';



ExecuteSkill.Parameter[2].ID := 2;
ExecuteSkill.Parameter[2].Name := 'TargetPosition Z';
ExecuteSkill.Parameter[2].Value := ZInputOutput;// ZCookieModule - ZCookieModuleCalibration - 2* Cookiethickness + toppingthickness+ Preasureheight  ;



(* ExecuteSkill.Parameter[4].ID := 4;
ExecuteSkill.Parameter[4].Name := 'Acceleration';
ExecuteSkill.Parameter[4].Value :=0 ;

*)
(*
ExecuteSkill.Parameter[5].ID := ;
ExecuteSkill.Parameter[5].Name := '';
ExecuteSkill.Parameter[5].Value := ;
*)



ExecuteSkill();

StepDone := ExecuteSkill.Done;
END_ACTION

ACTION ST31_BlockPump_active:
//RT: 2014.11.23: Blockirt den Mover an Position
StepDone := FALSE;

//Skill auswählen
ExecuteSkill.SkillID 		:= 1315;
ExecuteSkill.SkillName	 	:= 'Block';

//Parameter setzen

ExecuteSkill.Parameter[1].ID := 1;
ExecuteSkill.Parameter[1].Name := 'TaskID';
ExecuteSkill.Parameter[1].Value := Order.TaskID;


(*
ExecuteSkill.Parameter[2].ID := ;
ExecuteSkill.Parameter[2].Name := '';
ExecuteSkill.Parameter[2].Value := ;
*)

(*
ExecuteSkill.Parameter[3].ID := ;
ExecuteSkill.Parameter[3].Name := '';
ExecuteSkill.Parameter[3].Value := ;
*)

(*
ExecuteSkill.Parameter[4].ID := ;
ExecuteSkill.Parameter[4].Name := '';
ExecuteSkill.Parameter[4].Value := ;
*)

(*
ExecuteSkill.Parameter[5].ID := ;
ExecuteSkill.Parameter[5].Name := '';
ExecuteSkill.Parameter[5].Value := ;
*)



ExecuteSkill();

StepDone := ExecuteSkill.Done;
END_ACTION

ACTION ST12_Input_active:
//RT: 2014.11.23: Input Modul auslösen
StepDone := FALSE;

//Skill auswählen
ExecuteSkill.SkillID 		:= 1402;
ExecuteSkill.SkillName	 	:= 'Input';

//Parameter setzen

ExecuteSkill.Parameter[1].ID := 1;
ExecuteSkill.Parameter[1].Name := 'TaskID';
ExecuteSkill.Parameter[1].Value := Order.TaskID;


(*
ExecuteSkill.Parameter[2].ID := ;
ExecuteSkill.Parameter[2].Name := '';
ExecuteSkill.Parameter[2].Value := ;
*)

(*
ExecuteSkill.Parameter[3].ID := ;
ExecuteSkill.Parameter[3].Name := '';
ExecuteSkill.Parameter[3].Value := ;
*)

(*
ExecuteSkill.Parameter[4].ID := ;
ExecuteSkill.Parameter[4].Name := '';
ExecuteSkill.Parameter[4].Value := ;
*)

(*
ExecuteSkill.Parameter[5].ID := ;
ExecuteSkill.Parameter[5].Name := '';
ExecuteSkill.Parameter[5].Value := ;
*)



ExecuteSkill();

StepDone := ExecuteSkill.Done;
END_ACTION

ACTION ST14_Exit_active:
SectionReady := TRUE;
END_ACTION

ACTION ST33_UnblockPump_active:
//RT: 2014.11.23: Gibt Mover Position Frei
StepDone := FALSE;

//Skill auswählen
ExecuteSkill.SkillID 		:= 1316;
ExecuteSkill.SkillName	 	:= 'Unblock';

//Parameter setzen

ExecuteSkill.Parameter[1].ID := 1;
ExecuteSkill.Parameter[1].Name := 'TaskID';
ExecuteSkill.Parameter[1].Value := Order.TaskID;


(*
ExecuteSkill.Parameter[2].ID := ;
ExecuteSkill.Parameter[2].Name := '';
ExecuteSkill.Parameter[2].Value := ;
*)

(*
ExecuteSkill.Parameter[3].ID := ;
ExecuteSkill.Parameter[3].Name := '';
ExecuteSkill.Parameter[3].Value := ;
*)

(*
ExecuteSkill.Parameter[4].ID := ;
ExecuteSkill.Parameter[4].Name := '';
ExecuteSkill.Parameter[4].Value := ;
*)

(*
ExecuteSkill.Parameter[5].ID := ;
ExecuteSkill.Parameter[5].Name := '';
ExecuteSkill.Parameter[5].Value := ;
*)



ExecuteSkill();

StepDone := ExecuteSkill.Done;
END_ACTION

ACTION ST6_Completed_active:
//RT: 2014.11.23: Warte auf Execute = False
RecipeDone := TRUE;
StepDone := FALSE;
END_ACTION

ACTION ST3_Pump_active:
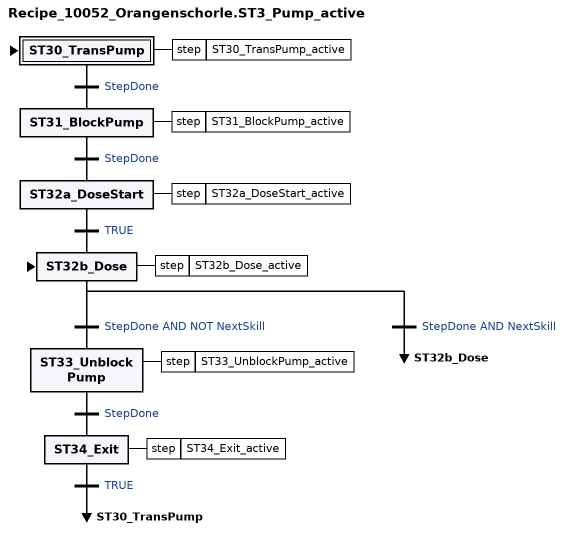
INITIAL_STEP ST30_TransPump:
    ST30_TransPump_active(N);  // step action
END_STEP
TRANSITION FROM ST30_TransPump TO ST31_BlockPump
    := StepDone;
END_TRANSITION
STEP ST31_BlockPump:
    ST31_BlockPump_active(N);  // step action
END_STEP
TRANSITION FROM ST31_BlockPump TO ST32a_DoseStart
    := StepDone;
END_TRANSITION
STEP ST32a_DoseStart:
    ST32a_DoseStart_active(N);  // step action
END_STEP
TRANSITION FROM ST32a_DoseStart TO ST32b_Dose
    := TRUE;
END_TRANSITION
STEP ST32b_Dose:
    ST32b_Dose_active(N);  // step action
END_STEP
TRANSITION FROM ST32b_Dose TO ST33_UnblockPump
    := StepDone AND NOT NextSkill;
END_TRANSITION
STEP ST33_UnblockPump:
    ST33_UnblockPump_active(N);  // step action
END_STEP
TRANSITION FROM ST33_UnblockPump TO ST34_Exit
    := StepDone;
END_TRANSITION
STEP ST34_Exit:
    ST34_Exit_active(N);  // step action
END_STEP
TRANSITION FROM ST34_Exit TO ST30_TransPump
    := TRUE;
END_TRANSITION
TRANSITION FROM ST32b_Dose TO ST32b_Dose
    := StepDone AND NextSkill;
END_TRANSITION
END_ACTION

ACTION ST10_TransToInput_active:
//RT: 2014.11.23: Mover zum Input

StepDone := FALSE;

//Skill auswählen
ExecuteSkill.SkillID 		:= 1320;
ExecuteSkill.SkillName	 	:= 'Transport';

//Parameter setzen

ExecuteSkill.Parameter[3].ID := 3;
ExecuteSkill.Parameter[3].Name := 'Velocity';
ExecuteSkill.Parameter[3].Value := 1000;



ExecuteSkill.Parameter[1].ID :=  1;
ExecuteSkill.Parameter[1].Name := 'TargetPosition X';
ExecuteSkill.Parameter[1].Value := 30 ;
ExecuteSkill.Parameter[1].StringValue := '#DP#2#XPosition';



ExecuteSkill.Parameter[2].ID := 2;
ExecuteSkill.Parameter[2].Name := 'TargetPosition Z';
ExecuteSkill.Parameter[2].Value := 100;// ZCookieModule - ZCookieModuleCalibration - 2* Cookiethickness + toppingthickness+ Preasureheight  ;



(*
ExecuteSkill.Parameter[4].ID := 4;
ExecuteSkill.Parameter[4].Name := 'Acceleration';
ExecuteSkill.Parameter[4].Value := 0 ;
*)

(*
ExecuteSkill.Parameter[5].ID := ;
ExecuteSkill.Parameter[5].Name := '';
ExecuteSkill.Parameter[5].Value := ;
*)



ExecuteSkill();

StepDone := ExecuteSkill.Done;
END_ACTION

ACTION ST34_Exit_active:
SectionReady := TRUE;
END_ACTION

ACTION ST32b_Dose_exit:

END_ACTION

ACTION ST42_CocktailOutput_active:
//RT: 2014.11.23: Ausgeben des Produktes
StepDone := FALSE;

//Skill auswählen
ExecuteSkill.SkillID 		:= 1403;
ExecuteSkill.SkillName	 	:= 'Output';

//Parameter setzen

ExecuteSkill.Parameter[1].ID := 1;
ExecuteSkill.Parameter[1].Name := 'TaskID';
ExecuteSkill.Parameter[1].Value := Order.TaskID;


(*
ExecuteSkill.Parameter[2].ID := ;
ExecuteSkill.Parameter[2].Name := '';
ExecuteSkill.Parameter[2].Value := ;
*)

(*
ExecuteSkill.Parameter[3].ID := ;
ExecuteSkill.Parameter[3].Name := '';
ExecuteSkill.Parameter[3].Value := ;
*)

(*
ExecuteSkill.Parameter[4].ID := ;
ExecuteSkill.Parameter[4].Name := '';
ExecuteSkill.Parameter[4].Value := ;
*)

(*
ExecuteSkill.Parameter[5].ID := ;
ExecuteSkill.Parameter[5].Name := '';
ExecuteSkill.Parameter[5].Value := ;
*)



ExecuteSkill();

StepDone := ExecuteSkill.Done;
END_ACTION

ACTION ST32a_DoseStart_active:
//RT: 2014.11.23: Summe aller zutaten zum Normiren

userparametersum := 0;
FOR i := 1 TO UserParameterCnt DO
	IF NOT (order.UserParameter[i].Value = 0) THEN
		userparametersum := userparametersum + order.UserParameter[i].Value;
	
	END_IF
END_FOR
IF userparametersum = 0 THEN
userparametersum := -1;
END_IF

//RT: 2014.11.23: Start wert des Arrays setzen
i := 1;
NextSkill := TRUE ;
END_ACTION

ACTION ST41_BlockOutput_active:
//RT: 2014.11.23: Blockirt den Mover an Position
StepDone := FALSE;

//Skill auswählen
ExecuteSkill.SkillID 		:= 1315;
ExecuteSkill.SkillName	 	:= 'Block';

//Parameter setzen

ExecuteSkill.Parameter[1].ID := 1;
ExecuteSkill.Parameter[1].Name := 'TaskID';
ExecuteSkill.Parameter[1].Value := Order.TaskID;


(*
ExecuteSkill.Parameter[2].ID := ;
ExecuteSkill.Parameter[2].Name := '';
ExecuteSkill.Parameter[2].Value := ;
*)

(*
ExecuteSkill.Parameter[3].ID := ;
ExecuteSkill.Parameter[3].Name := '';
ExecuteSkill.Parameter[3].Value := ;
*)

(*
ExecuteSkill.Parameter[4].ID := ;
ExecuteSkill.Parameter[4].Name := '';
ExecuteSkill.Parameter[4].Value := ;
*)

(*
ExecuteSkill.Parameter[5].ID := ;
ExecuteSkill.Parameter[5].Name := '';
ExecuteSkill.Parameter[5].Value := ;
*)



ExecuteSkill();

StepDone := ExecuteSkill.Done;
END_ACTION

ACTION ST4_Output_entry:
SectionReady := FALSE;
END_ACTION

ACTION ST44_Exit_active:
SectionReady := TRUE;
END_ACTION

END_FUNCTION_BLOCK

// ---- POUs/Recipes/Recipe_10054_Sixteen.TcPOU
FUNCTION_BLOCK Recipe_10054_Sixteen
VAR_INPUT
	execute: BOOL;
	Order: DUT_RECIPEORDER;
END_VAR
VAR_OUTPUT
	RecipeInfo: DUT_RECIPEOFFER;
	RecipeDone: BOOL;
	InitDone: BOOL;
	Ready: BOOL;
END_VAR
VAR
	userparametersum: LREAL;
	StepDone: BOOL;
	i: INT;
	Command: ARRAY[1..5] OF DUT_RecipeCommand;
	NextSkill: BOOL;
	SectionReady: BOOL;
END_VAR

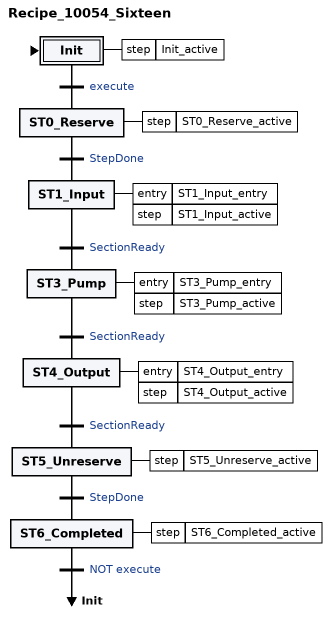
INITIAL_STEP Init:
    Init_active(N);  // step action
END_STEP
TRANSITION FROM Init TO ST0_Reserve
    := execute;
END_TRANSITION
STEP ST0_Reserve:
    ST0_Reserve_active(N);  // step action
END_STEP
TRANSITION FROM ST0_Reserve TO ST1_Input
    := StepDone;
END_TRANSITION
STEP ST1_Input:
    ST1_Input_entry(P1);  // entry action
    ST1_Input_active(N);  // step action
END_STEP
TRANSITION FROM ST1_Input TO ST3_Pump
    := SectionReady;
END_TRANSITION
STEP ST3_Pump:
    ST3_Pump_entry(P1);  // entry action
    ST3_Pump_active(N);  // step action
END_STEP
TRANSITION FROM ST3_Pump TO ST4_Output
    := SectionReady;
END_TRANSITION
STEP ST4_Output:
    ST4_Output_entry(P1);  // entry action
    ST4_Output_active(N);  // step action
END_STEP
TRANSITION FROM ST4_Output TO ST5_Unreserve
    := SectionReady;
END_TRANSITION
STEP ST5_Unreserve:
    ST5_Unreserve_active(N);  // step action
END_STEP
TRANSITION FROM ST5_Unreserve TO ST6_Completed
    := StepDone;
END_TRANSITION
STEP ST6_Completed:
    ST6_Completed_active(N);  // step action
END_STEP
TRANSITION FROM ST6_Completed TO Init
    := NOT execute;
END_TRANSITION

ACTION ST32b_Dose_exit:

END_ACTION

ACTION ST40_TransOutput_active:
//RT: 2014.11.23: Mover zum Output
StepDone := FALSE;

//Skill auswählen
ExecuteSkill.SkillID 		:= 1320;
ExecuteSkill.SkillName	 	:= 'Transport';

//Parameter setzen

ExecuteSkill.Parameter[3].ID := 3;
ExecuteSkill.Parameter[3].Name := 'Velocity';
ExecuteSkill.Parameter[3].Value := 300;



ExecuteSkill.Parameter[1].ID :=  1;
ExecuteSkill.Parameter[1].Name := 'TargetPosition X';
ExecuteSkill.Parameter[1].Value := 30 ;
ExecuteSkill.Parameter[1].StringValue := '#DP#2#XPosition';



ExecuteSkill.Parameter[2].ID := 2;
ExecuteSkill.Parameter[2].Name := 'TargetPosition Z';
ExecuteSkill.Parameter[2].Value := 100;// ZCookieModule - ZCookieModuleCalibration - 2* Cookiethickness + toppingthickness+ Preasureheight  ;



(* ExecuteSkill.Parameter[4].ID := 4;
ExecuteSkill.Parameter[4].Name := 'Acceleration';
ExecuteSkill.Parameter[4].Value :=0 ;

*)
(*
ExecuteSkill.Parameter[5].ID := ;
ExecuteSkill.Parameter[5].Name := '';
ExecuteSkill.Parameter[5].Value := ;
*)



ExecuteSkill();

StepDone := ExecuteSkill.Done;
END_ACTION

ACTION ST12_Input_active:
//RT: 2014.11.23: Input Modul auslösen
StepDone := FALSE;

//Skill auswählen
ExecuteSkill.SkillID 		:= 1402;
ExecuteSkill.SkillName	 	:= 'Input';

//Parameter setzen

ExecuteSkill.Parameter[1].ID := 1;
ExecuteSkill.Parameter[1].Name := 'TaskID';
ExecuteSkill.Parameter[1].Value := Order.TaskID;


(*
ExecuteSkill.Parameter[2].ID := ;
ExecuteSkill.Parameter[2].Name := '';
ExecuteSkill.Parameter[2].Value := ;
*)

(*
ExecuteSkill.Parameter[3].ID := ;
ExecuteSkill.Parameter[3].Name := '';
ExecuteSkill.Parameter[3].Value := ;
*)

(*
ExecuteSkill.Parameter[4].ID := ;
ExecuteSkill.Parameter[4].Name := '';
ExecuteSkill.Parameter[4].Value := ;
*)

(*
ExecuteSkill.Parameter[5].ID := ;
ExecuteSkill.Parameter[5].Name := '';
ExecuteSkill.Parameter[5].Value := ;
*)



ExecuteSkill();

StepDone := ExecuteSkill.Done;
END_ACTION

ACTION ST13_UnblockInput_active:
//RT: 2014.11.23: Gibt Mover Position Frei
StepDone := FALSE;

//Skill auswählen
ExecuteSkill.SkillID 		:= 1316;
ExecuteSkill.SkillName	 	:= 'Unblock';

//Parameter setzen

ExecuteSkill.Parameter[1].ID := 1;
ExecuteSkill.Parameter[1].Name := 'TaskID';
ExecuteSkill.Parameter[1].Value := Order.TaskID;


(*
ExecuteSkill.Parameter[2].ID := ;
ExecuteSkill.Parameter[2].Name := '';
ExecuteSkill.Parameter[2].Value := ;
*)

(*
ExecuteSkill.Parameter[3].ID := ;
ExecuteSkill.Parameter[3].Name := '';
ExecuteSkill.Parameter[3].Value := ;
*)

(*
ExecuteSkill.Parameter[4].ID := ;
ExecuteSkill.Parameter[4].Name := '';
ExecuteSkill.Parameter[4].Value := ;
*)

(*
ExecuteSkill.Parameter[5].ID := ;
ExecuteSkill.Parameter[5].Name := '';
ExecuteSkill.Parameter[5].Value := ;
*)



ExecuteSkill();

StepDone := ExecuteSkill.Done;
END_ACTION

ACTION ST42_CocktailOutput_active:
//RT: 2014.11.23: Ausgeben des Produktes
StepDone := FALSE;

//Skill auswählen
ExecuteSkill.SkillID 		:= 1403;
ExecuteSkill.SkillName	 	:= 'Output';

//Parameter setzen

ExecuteSkill.Parameter[1].ID := 1;
ExecuteSkill.Parameter[1].Name := 'TaskID';
ExecuteSkill.Parameter[1].Value := Order.TaskID;


(*
ExecuteSkill.Parameter[2].ID := ;
ExecuteSkill.Parameter[2].Name := '';
ExecuteSkill.Parameter[2].Value := ;
*)

(*
ExecuteSkill.Parameter[3].ID := ;
ExecuteSkill.Parameter[3].Name := '';
ExecuteSkill.Parameter[3].Value := ;
*)

(*
ExecuteSkill.Parameter[4].ID := ;
ExecuteSkill.Parameter[4].Name := '';
ExecuteSkill.Parameter[4].Value := ;
*)

(*
ExecuteSkill.Parameter[5].ID := ;
ExecuteSkill.Parameter[5].Name := '';
ExecuteSkill.Parameter[5].Value := ;
*)



ExecuteSkill();

StepDone := ExecuteSkill.Done;
END_ACTION

ACTION ST6_Completed_active:
//RT: 2014.11.23: Warte auf Execute = False
RecipeDone := TRUE;
StepDone := FALSE;
END_ACTION

ACTION ST4_Output_entry:
SectionReady := FALSE;
END_ACTION

ACTION ST44_Exit_active:
SectionReady := TRUE;
END_ACTION

ACTION ST4_Output_active:
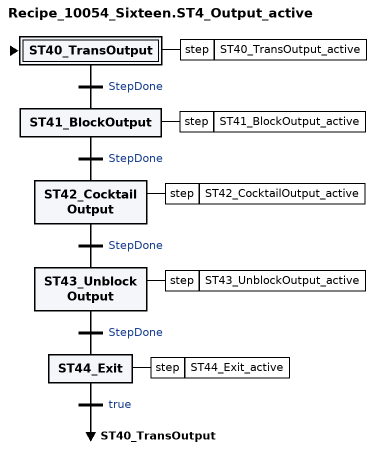
INITIAL_STEP ST40_TransOutput:
    ST40_TransOutput_active(N);  // step action
END_STEP
TRANSITION FROM ST40_TransOutput TO ST41_BlockOutput
    := StepDone;
END_TRANSITION
STEP ST41_BlockOutput:
    ST41_BlockOutput_active(N);  // step action
END_STEP
TRANSITION FROM ST41_BlockOutput TO ST42_CocktailOutput
    := StepDone;
END_TRANSITION
STEP ST42_CocktailOutput:
    ST42_CocktailOutput_active(N);  // step action
END_STEP
TRANSITION FROM ST42_CocktailOutput TO ST43_UnblockOutput
    := StepDone;
END_TRANSITION
STEP ST43_UnblockOutput:
    ST43_UnblockOutput_active(N);  // step action
END_STEP
TRANSITION FROM ST43_UnblockOutput TO ST44_Exit
    := StepDone;
END_TRANSITION
STEP ST44_Exit:
    ST44_Exit_active(N);  // step action
END_STEP
TRANSITION FROM ST44_Exit TO ST40_TransOutput
    := true;
END_TRANSITION
END_ACTION

ACTION Init_active:
//RT: 2014.11.23: Vorbereiten der daten und der HMI
RecipeDone := FALSE;

// Initialisation of Recipe Parameters an name etc
RecipeInfo.Name := 'Sixteen';
RecipeInfo.Description := '';
RecipeInfo.Dummy := FALSE;
RecipeInfo.RecipeID := 10054; 	// 
Initdone := TRUE;

//RT: 2014.11.23: wenn weniger als 5 alle lehren skills SkillID := 0
Command[1].SkillID := 1111;
Command[1].SkillName := 'Grenadine Syrup';
Command[1].Quantity := 11;

Command[2].SkillID := 1112;
Command[2].SkillName := 'Lemon Juice';
Command[2].Quantity := 11;

Command[3].SkillID := 1114;
Command[3].SkillName := 'Pineapple Juice';
Command[3].Quantity := 22;

Command[4].SkillID := 1117;
Command[4].SkillName := 'Orange Juice';
Command[4].Quantity := 45;

Command[5].SkillID := 1113;
Command[5].SkillName := 'Maracuja Juice';
Command[5].Quantity := 11;








//Parameter 0:

	RecipeInfo.UserParameter[0].Dummy 		:= FALSE;
	RecipeInfo.UserParameter[0].Default		:= 200;
	RecipeInfo.UserParameter[0].Description	:= 'Gives the total fluid amount in the glass';
	RecipeInfo.UserParameter[0].MaxValue	:= 200;
	RecipeInfo.UserParameter[0].MinValue	:= 10;
	RecipeInfo.UserParameter[0].Name		:= 'Total Liquid Amount';
	RecipeInfo.UserParameter[0].Unit		:= 'ml';
	
//Parameter 1-5:
FOR i := 1 TO 5 DO
	IF Command[i].SkillID = 0 THEN
		RecipeInfo.UserParameter[i].Dummy 		:= TRUE;
	ELSE
		RecipeInfo.UserParameter[i].Dummy 		:= FALSE;
		RecipeInfo.UserParameter[i].Default		:= Command[i].Quantity;
		RecipeInfo.UserParameter[i].Description	:= Command[i].SkillName;
		RecipeInfo.UserParameter[i].MaxValue	:= 100;
		RecipeInfo.UserParameter[i].MinValue	:= 1;
		RecipeInfo.UserParameter[i].Name		:= Command[i].SkillName;
		RecipeInfo.UserParameter[i].Unit		:= 'ml';	
	END_IF
END_FOR
END_ACTION

ACTION ST3_Pump_active:
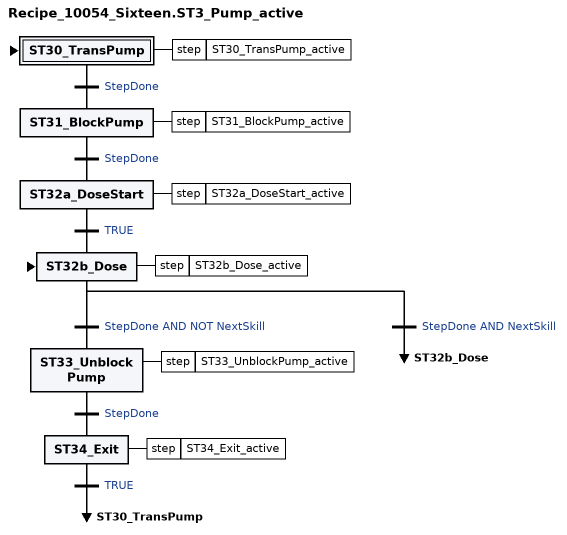
INITIAL_STEP ST30_TransPump:
    ST30_TransPump_active(N);  // step action
END_STEP
TRANSITION FROM ST30_TransPump TO ST31_BlockPump
    := StepDone;
END_TRANSITION
STEP ST31_BlockPump:
    ST31_BlockPump_active(N);  // step action
END_STEP
TRANSITION FROM ST31_BlockPump TO ST32a_DoseStart
    := StepDone;
END_TRANSITION
STEP ST32a_DoseStart:
    ST32a_DoseStart_active(N);  // step action
END_STEP
TRANSITION FROM ST32a_DoseStart TO ST32b_Dose
    := TRUE;
END_TRANSITION
STEP ST32b_Dose:
    ST32b_Dose_active(N);  // step action
END_STEP
TRANSITION FROM ST32b_Dose TO ST33_UnblockPump
    := StepDone AND NOT NextSkill;
END_TRANSITION
STEP ST33_UnblockPump:
    ST33_UnblockPump_active(N);  // step action
END_STEP
TRANSITION FROM ST33_UnblockPump TO ST34_Exit
    := StepDone;
END_TRANSITION
STEP ST34_Exit:
    ST34_Exit_active(N);  // step action
END_STEP
TRANSITION FROM ST34_Exit TO ST30_TransPump
    := TRUE;
END_TRANSITION
TRANSITION FROM ST32b_Dose TO ST32b_Dose
    := StepDone AND NextSkill;
END_TRANSITION
END_ACTION

ACTION ST34_Exit_active:
SectionReady := TRUE;
END_ACTION

ACTION ST10_TransToInput_active:
//RT: 2014.11.23: Mover zum Input

StepDone := FALSE;

//Skill auswählen
ExecuteSkill.SkillID 		:= 1320;
ExecuteSkill.SkillName	 	:= 'Transport';

//Parameter setzen

ExecuteSkill.Parameter[3].ID := 3;
ExecuteSkill.Parameter[3].Name := 'Velocity';
ExecuteSkill.Parameter[3].Value := 1000;



ExecuteSkill.Parameter[1].ID :=  1;
ExecuteSkill.Parameter[1].Name := 'TargetPosition X';
ExecuteSkill.Parameter[1].Value := 30 ;
ExecuteSkill.Parameter[1].StringValue := '#DP#2#XPosition';



ExecuteSkill.Parameter[2].ID := 2;
ExecuteSkill.Parameter[2].Name := 'TargetPosition Z';
ExecuteSkill.Parameter[2].Value := 100;// ZCookieModule - ZCookieModuleCalibration - 2* Cookiethickness + toppingthickness+ Preasureheight  ;



(*
ExecuteSkill.Parameter[4].ID := 4;
ExecuteSkill.Parameter[4].Name := 'Acceleration';
ExecuteSkill.Parameter[4].Value := 0 ;
*)

(*
ExecuteSkill.Parameter[5].ID := ;
ExecuteSkill.Parameter[5].Name := '';
ExecuteSkill.Parameter[5].Value := ;
*)



ExecuteSkill();

StepDone := ExecuteSkill.Done;
END_ACTION

ACTION ST1_Input_entry:
SectionReady := FALSE;
END_ACTION

ACTION ST32b_Dose_active:
//RT: 2014.11.23: Die Dosir Skills anlegen
StepDone := FALSE;

//Skill auswählen
ExecuteSkill.SkillID 		:= Command[i].SkillID;
ExecuteSkill.SkillName	 	:= Command[i].SkillName;
//Parameter setzen

ExecuteSkill.Parameter[0].ID := 1;
ExecuteSkill.Parameter[0].Name := 'Quantity';
//order.userParameter[0] = amount
ExecuteSkill.Parameter[0].Value := order.UserParameter[0].Value * order.UserParameter[i].Value / userparametersum ;//Summe aller Zutatenmengen;

(*
ExecuteSkill.Parameter[2].ID := ;
ExecuteSkill.Parameter[2].Name := '';
ExecuteSkill.Parameter[2].Value := ;
*)

(*
ExecuteSkill.Parameter[3].ID := ;
ExecuteSkill.Parameter[3].Name := '';
ExecuteSkill.Parameter[3].Value := ;
*)

(*
ExecuteSkill.Parameter[4].ID := ;
ExecuteSkill.Parameter[4].Name := '';
ExecuteSkill.Parameter[4].Value := ;
*)

(*
ExecuteSkill.Parameter[5].ID := ;
ExecuteSkill.Parameter[5].Name := '';
ExecuteSkill.Parameter[5].Value := ;
*)


ExecuteSkill();

StepDone := ExecuteSkill.Done;

i := i + 1 ;

IF i = 6 THEN
	NextSkill := FALSE;
ELSIF Command[i].SkillID = 0 THEN
	NextSkill := FALSE;
ELSE
	NextSkill := TRUE;
END_IF
END_ACTION

ACTION ST3_Pump_entry:
SectionReady := FALSE;
END_ACTION

ACTION ST43_UnblockOutput_active:
//RT: 2014.11.23: Gibt Mover Position Frei
StepDone := FALSE;

//Skill auswählen
ExecuteSkill.SkillID 		:= 1316;
ExecuteSkill.SkillName	 	:= 'Unblock';

//Parameter setzen

ExecuteSkill.Parameter[1].ID := 1;
ExecuteSkill.Parameter[1].Name := 'TaskID';
ExecuteSkill.Parameter[1].Value := Order.TaskID;


(*
ExecuteSkill.Parameter[2].ID := ;
ExecuteSkill.Parameter[2].Name := '';
ExecuteSkill.Parameter[2].Value := ;
*)

(*
ExecuteSkill.Parameter[3].ID := ;
ExecuteSkill.Parameter[3].Name := '';
ExecuteSkill.Parameter[3].Value := ;
*)

(*
ExecuteSkill.Parameter[4].ID := ;
ExecuteSkill.Parameter[4].Name := '';
ExecuteSkill.Parameter[4].Value := ;
*)

(*
ExecuteSkill.Parameter[5].ID := ;
ExecuteSkill.Parameter[5].Name := '';
ExecuteSkill.Parameter[5].Value := ;
*)



ExecuteSkill();

StepDone := ExecuteSkill.Done;
END_ACTION

ACTION ST1_Input_active:
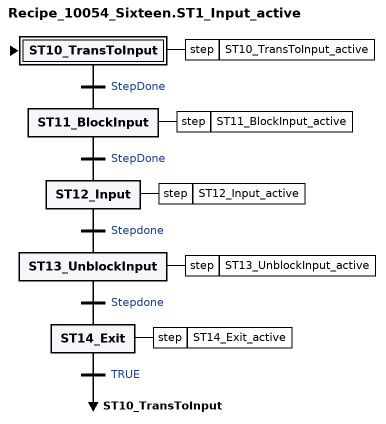
INITIAL_STEP ST10_TransToInput:
    ST10_TransToInput_active(N);  // step action
END_STEP
TRANSITION FROM ST10_TransToInput TO ST11_BlockInput
    := StepDone;
END_TRANSITION
STEP ST11_BlockInput:
    ST11_BlockInput_active(N);  // step action
END_STEP
TRANSITION FROM ST11_BlockInput TO ST12_Input
    := StepDone;
END_TRANSITION
STEP ST12_Input:
    ST12_Input_active(N);  // step action
END_STEP
TRANSITION FROM ST12_Input TO ST13_UnblockInput
    := Stepdone;
END_TRANSITION
STEP ST13_UnblockInput:
    ST13_UnblockInput_active(N);  // step action
END_STEP
TRANSITION FROM ST13_UnblockInput TO ST14_Exit
    := Stepdone;
END_TRANSITION
STEP ST14_Exit:
    ST14_Exit_active(N);  // step action
END_STEP
TRANSITION FROM ST14_Exit TO ST10_TransToInput
    := TRUE;
END_TRANSITION
END_ACTION

ACTION ST1_Reserve0_active:
//RT: 2014.11.23: Reservire einen Mover

StepDone := FALSE;
RecipeDone := FALSE;
//Skill auswählen
ExecuteSkill.SkillID 		:= 1310;
ExecuteSkill.SkillName	 	:= 'Reserve';

//Parameter setzen

ExecuteSkill.Parameter[1].ID := 1;
ExecuteSkill.Parameter[1].Name := 'TaskID';
ExecuteSkill.Parameter[1].Value := Order.TaskID;

(*
ExecuteSkill.Parameter[2].ID := ;
ExecuteSkill.Parameter[2].Name := '';
ExecuteSkill.Parameter[2].Value := ;
*)

(*
ExecuteSkill.Parameter[3].ID := ;
ExecuteSkill.Parameter[3].Name := '';
ExecuteSkill.Parameter[3].Value := ;
*)

(*
ExecuteSkill.Parameter[4].ID := ;
ExecuteSkill.Parameter[4].Name := '';
ExecuteSkill.Parameter[4].Value := ;
*)

(*
ExecuteSkill.Parameter[5].ID := ;
ExecuteSkill.Parameter[5].Name := '';
ExecuteSkill.Parameter[5].Value := ;
*)

ExecuteSkill();

StepDone := ExecuteSkill.Done;
END_ACTION

ACTION ST32a_DoseStart_active:
//RT: 2014.11.23: Summe aller zutaten zum Normiren

userparametersum := 0;
FOR i := 1 TO UserParameterCnt DO
	IF NOT (order.UserParameter[i].Value = 0) THEN
		userparametersum := userparametersum + order.UserParameter[i].Value;
	
	END_IF
END_FOR
IF userparametersum = 0 THEN
userparametersum := -1;
END_IF

//RT: 2014.11.23: Start wert des Arrays setzen
i := 1;
NextSkill := TRUE ;
END_ACTION

ACTION ST0_Reserve_active:
//RT: 2014.11.23: Reservire einen Mover

StepDone := FALSE;
RecipeDone := FALSE;
//Skill auswählen
ExecuteSkill.SkillID 		:= 1310;
ExecuteSkill.SkillName	 	:= 'Reserve';

//Parameter setzen

ExecuteSkill.Parameter[1].ID := 1;
ExecuteSkill.Parameter[1].Name := 'TaskID';
ExecuteSkill.Parameter[1].Value := Order.TaskID;

(*
ExecuteSkill.Parameter[2].ID := ;
ExecuteSkill.Parameter[2].Name := '';
ExecuteSkill.Parameter[2].Value := ;
*)

(*
ExecuteSkill.Parameter[3].ID := ;
ExecuteSkill.Parameter[3].Name := '';
ExecuteSkill.Parameter[3].Value := ;
*)

(*
ExecuteSkill.Parameter[4].ID := ;
ExecuteSkill.Parameter[4].Name := '';
ExecuteSkill.Parameter[4].Value := ;
*)

(*
ExecuteSkill.Parameter[5].ID := ;
ExecuteSkill.Parameter[5].Name := '';
ExecuteSkill.Parameter[5].Value := ;
*)

ExecuteSkill();

StepDone := ExecuteSkill.Done;
END_ACTION

ACTION ST5_Unreserve_active:
//RT: 2014.11.23: Mover Freigeben
StepDone := FALSE;

//Skill auswählen
ExecuteSkill.SkillID 		:= 1311;
ExecuteSkill.SkillName	 	:= 'Unreserve';

//Parameter setzen

ExecuteSkill.Parameter[1].ID := 1;
ExecuteSkill.Parameter[1].Name := 'TaskID';
ExecuteSkill.Parameter[1].Value := Order.TaskID;


(*
ExecuteSkill.Parameter[2].ID := ;
ExecuteSkill.Parameter[2].Name := '';
ExecuteSkill.Parameter[2].Val ue := ;
*)

(*
ExecuteSkill.Parameter[3].ID := ;
ExecuteSkill.Parameter[3].Name := '';
ExecuteSkill.Parameter[3].Value := ;
*)

(*
ExecuteSkill.Parameter[4].ID := ;
ExecuteSkill.Parameter[4].Name := '';
ExecuteSkill.Parameter[4].Value := ;
*)

(*
ExecuteSkill.Parameter[5].ID := ;
ExecuteSkill.Parameter[5].Name := '';
ExecuteSkill.Parameter[5].Value := ;
*)



ExecuteSkill();

StepDone := ExecuteSkill.Done;
END_ACTION

ACTION ST31_BlockPump_active:
//RT: 2014.11.23: Blockirt den Mover an Position
StepDone := FALSE;

//Skill auswählen
ExecuteSkill.SkillID 		:= 1315;
ExecuteSkill.SkillName	 	:= 'Block';

//Parameter setzen

ExecuteSkill.Parameter[1].ID := 1;
ExecuteSkill.Parameter[1].Name := 'TaskID';
ExecuteSkill.Parameter[1].Value := Order.TaskID;


(*
ExecuteSkill.Parameter[2].ID := ;
ExecuteSkill.Parameter[2].Name := '';
ExecuteSkill.Parameter[2].Value := ;
*)

(*
ExecuteSkill.Parameter[3].ID := ;
ExecuteSkill.Parameter[3].Name := '';
ExecuteSkill.Parameter[3].Value := ;
*)

(*
ExecuteSkill.Parameter[4].ID := ;
ExecuteSkill.Parameter[4].Name := '';
ExecuteSkill.Parameter[4].Value := ;
*)

(*
ExecuteSkill.Parameter[5].ID := ;
ExecuteSkill.Parameter[5].Name := '';
ExecuteSkill.Parameter[5].Value := ;
*)



ExecuteSkill();

StepDone := ExecuteSkill.Done;
END_ACTION

ACTION ST14_Exit_active:
SectionReady := TRUE;
END_ACTION

ACTION ST41_BlockOutput_active:
//RT: 2014.11.23: Blockirt den Mover an Position
StepDone := FALSE;

//Skill auswählen
ExecuteSkill.SkillID 		:= 1315;
ExecuteSkill.SkillName	 	:= 'Block';

//Parameter setzen

ExecuteSkill.Parameter[1].ID := 1;
ExecuteSkill.Parameter[1].Name := 'TaskID';
ExecuteSkill.Parameter[1].Value := Order.TaskID;


(*
ExecuteSkill.Parameter[2].ID := ;
ExecuteSkill.Parameter[2].Name := '';
ExecuteSkill.Parameter[2].Value := ;
*)

(*
ExecuteSkill.Parameter[3].ID := ;
ExecuteSkill.Parameter[3].Name := '';
ExecuteSkill.Parameter[3].Value := ;
*)

(*
ExecuteSkill.Parameter[4].ID := ;
ExecuteSkill.Parameter[4].Name := '';
ExecuteSkill.Parameter[4].Value := ;
*)

(*
ExecuteSkill.Parameter[5].ID := ;
ExecuteSkill.Parameter[5].Name := '';
ExecuteSkill.Parameter[5].Value := ;
*)



ExecuteSkill();

StepDone := ExecuteSkill.Done;
END_ACTION

ACTION ST33_UnblockPump_active:
//RT: 2014.11.23: Gibt Mover Position Frei
StepDone := FALSE;

//Skill auswählen
ExecuteSkill.SkillID 		:= 1316;
ExecuteSkill.SkillName	 	:= 'Unblock';

//Parameter setzen

ExecuteSkill.Parameter[1].ID := 1;
ExecuteSkill.Parameter[1].Name := 'TaskID';
ExecuteSkill.Parameter[1].Value := Order.TaskID;


(*
ExecuteSkill.Parameter[2].ID := ;
ExecuteSkill.Parameter[2].Name := '';
ExecuteSkill.Parameter[2].Value := ;
*)

(*
ExecuteSkill.Parameter[3].ID := ;
ExecuteSkill.Parameter[3].Name := '';
ExecuteSkill.Parameter[3].Value := ;
*)

(*
ExecuteSkill.Parameter[4].ID := ;
ExecuteSkill.Parameter[4].Name := '';
ExecuteSkill.Parameter[4].Value := ;
*)

(*
ExecuteSkill.Parameter[5].ID := ;
ExecuteSkill.Parameter[5].Name := '';
ExecuteSkill.Parameter[5].Value := ;
*)



ExecuteSkill();

StepDone := ExecuteSkill.Done;
END_ACTION

ACTION ST11_BlockInput_active:
//RT: 2014.11.23: Blockirt den Mover an Position
StepDone := FALSE;

//Skill auswählen
ExecuteSkill.SkillID 		:= 1315;
ExecuteSkill.SkillName	 	:= 'Block';

//Parameter setzen

ExecuteSkill.Parameter[1].ID := 1;
ExecuteSkill.Parameter[1].Name := 'TaskID';
ExecuteSkill.Parameter[1].Value := Order.TaskID;


(*
ExecuteSkill.Parameter[2].ID := ;
ExecuteSkill.Parameter[2].Name := '';
ExecuteSkill.Parameter[2].Value := ;
*)

(*
ExecuteSkill.Parameter[3].ID := ;
ExecuteSkill.Parameter[3].Name := '';
ExecuteSkill.Parameter[3].Value := ;
*)

(*
ExecuteSkill.Parameter[4].ID := ;
ExecuteSkill.Parameter[4].Name := '';
ExecuteSkill.Parameter[4].Value := ;
*)

(*
ExecuteSkill.Parameter[5].ID := ;
ExecuteSkill.Parameter[5].Name := '';
ExecuteSkill.Parameter[5].Value := ;
*)



ExecuteSkill();

StepDone := ExecuteSkill.Done;
END_ACTION

ACTION ST30_TransPump_active:
//RT: 2014.11.23: Mover zum Pump
StepDone := FALSE;

//Skill auswählen
ExecuteSkill.SkillID 		:= 1320;
ExecuteSkill.SkillName	 	:= 'Transport';

//Parameter setzen

ExecuteSkill.Parameter[3].ID := 3;
ExecuteSkill.Parameter[3].Name := 'Velocity';
ExecuteSkill.Parameter[3].Value := 1000;



ExecuteSkill.Parameter[1].ID :=  1;
ExecuteSkill.Parameter[1].Name := 'TargetPosition X';
ExecuteSkill.Parameter[1].Value := 30 ;
ExecuteSkill.Parameter[1].StringValue := '#DP#2#XPosition';



ExecuteSkill.Parameter[2].ID := 2;
ExecuteSkill.Parameter[2].Name := 'TargetPosition Z';
ExecuteSkill.Parameter[2].Value := 10;// ZCookieModule - ZCookieModuleCalibration - 2* Cookiethickness + toppingthickness+ Preasureheight  ;



(*
ExecuteSkill.Parameter[4].ID := 4;
ExecuteSkill.Parameter[4].Name := 'Acceleration';
ExecuteSkill.Parameter[4].Value := 0 ;
*)

(*
ExecuteSkill.Parameter[5].ID := ;
ExecuteSkill.Parameter[5].Name := '';
ExecuteSkill.Parameter[5].Value := ;
*)



ExecuteSkill();

StepDone := ExecuteSkill.Done;
END_ACTION

END_FUNCTION_BLOCK

// ---- POUs/Recipes/Recipe_10059_Pina_Batida_Lemon.TcPOU
FUNCTION_BLOCK Recipe_10059_Pina_Batida_Lemon
VAR_INPUT
	execute: BOOL;
	Order: DUT_RECIPEORDER;
END_VAR
VAR_OUTPUT
	RecipeInfo: DUT_RECIPEOFFER;
	RecipeDone: BOOL;
	InitDone: BOOL;
	Ready: BOOL;
END_VAR
VAR
	userparametersum: LREAL;
	StepDone: BOOL;
	i: INT;
	Command: ARRAY[1..5] OF DUT_RecipeCommand;
	NextSkill: BOOL;
	SectionReady: BOOL;
END_VAR

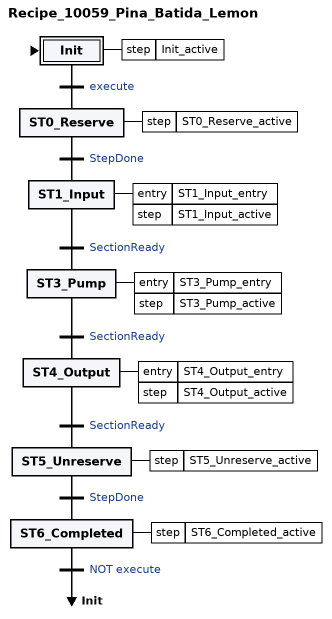
INITIAL_STEP Init:
    Init_active(N);  // step action
END_STEP
TRANSITION FROM Init TO ST0_Reserve
    := execute;
END_TRANSITION
STEP ST0_Reserve:
    ST0_Reserve_active(N);  // step action
END_STEP
TRANSITION FROM ST0_Reserve TO ST1_Input
    := StepDone;
END_TRANSITION
STEP ST1_Input:
    ST1_Input_entry(P1);  // entry action
    ST1_Input_active(N);  // step action
END_STEP
TRANSITION FROM ST1_Input TO ST3_Pump
    := SectionReady;
END_TRANSITION
STEP ST3_Pump:
    ST3_Pump_entry(P1);  // entry action
    ST3_Pump_active(N);  // step action
END_STEP
TRANSITION FROM ST3_Pump TO ST4_Output
    := SectionReady;
END_TRANSITION
STEP ST4_Output:
    ST4_Output_entry(P1);  // entry action
    ST4_Output_active(N);  // step action
END_STEP
TRANSITION FROM ST4_Output TO ST5_Unreserve
    := SectionReady;
END_TRANSITION
STEP ST5_Unreserve:
    ST5_Unreserve_active(N);  // step action
END_STEP
TRANSITION FROM ST5_Unreserve TO ST6_Completed
    := StepDone;
END_TRANSITION
STEP ST6_Completed:
    ST6_Completed_active(N);  // step action
END_STEP
TRANSITION FROM ST6_Completed TO Init
    := NOT execute;
END_TRANSITION

ACTION ST11_BlockInput_active:
//RT: 2014.11.23: Blockirt den Mover an Position
StepDone := FALSE;

//Skill auswählen
ExecuteSkill.SkillID 		:= 1315;
ExecuteSkill.SkillName	 	:= 'Block';

//Parameter setzen

ExecuteSkill.Parameter[1].ID := 1;
ExecuteSkill.Parameter[1].Name := 'TaskID';
ExecuteSkill.Parameter[1].Value := Order.TaskID;


(*
ExecuteSkill.Parameter[2].ID := ;
ExecuteSkill.Parameter[2].Name := '';
ExecuteSkill.Parameter[2].Value := ;
*)

(*
ExecuteSkill.Parameter[3].ID := ;
ExecuteSkill.Parameter[3].Name := '';
ExecuteSkill.Parameter[3].Value := ;
*)

(*
ExecuteSkill.Parameter[4].ID := ;
ExecuteSkill.Parameter[4].Name := '';
ExecuteSkill.Parameter[4].Value := ;
*)

(*
ExecuteSkill.Parameter[5].ID := ;
ExecuteSkill.Parameter[5].Name := '';
ExecuteSkill.Parameter[5].Value := ;
*)



ExecuteSkill();

StepDone := ExecuteSkill.Done;
END_ACTION

ACTION ST6_Completed_active:
//RT: 2014.11.23: Warte auf Execute = False
RecipeDone := TRUE;
StepDone := FALSE;
END_ACTION

ACTION ST32a_DoseStart_active:
//RT: 2014.11.23: Summe aller zutaten zum Normiren

userparametersum := 0;
FOR i := 1 TO UserParameterCnt DO
	IF NOT (order.UserParameter[i].Value = 0) THEN
		userparametersum := userparametersum + order.UserParameter[i].Value;
	
	END_IF
END_FOR
IF userparametersum = 0 THEN
userparametersum := -1;
END_IF

//RT: 2014.11.23: Start wert des Arrays setzen
i := 1;
NextSkill := TRUE ;
END_ACTION

ACTION ST32b_Dose_exit:

END_ACTION

ACTION ST12_Input_active:
//RT: 2014.11.23: Input Modul auslösen
StepDone := FALSE;

//Skill auswählen
ExecuteSkill.SkillID 		:= 1402;
ExecuteSkill.SkillName	 	:= 'Input';

//Parameter setzen

ExecuteSkill.Parameter[1].ID := 1;
ExecuteSkill.Parameter[1].Name := 'TaskID';
ExecuteSkill.Parameter[1].Value := Order.TaskID;


(*
ExecuteSkill.Parameter[2].ID := ;
ExecuteSkill.Parameter[2].Name := '';
ExecuteSkill.Parameter[2].Value := ;
*)

(*
ExecuteSkill.Parameter[3].ID := ;
ExecuteSkill.Parameter[3].Name := '';
ExecuteSkill.Parameter[3].Value := ;
*)

(*
ExecuteSkill.Parameter[4].ID := ;
ExecuteSkill.Parameter[4].Name := '';
ExecuteSkill.Parameter[4].Value := ;
*)

(*
ExecuteSkill.Parameter[5].ID := ;
ExecuteSkill.Parameter[5].Name := '';
ExecuteSkill.Parameter[5].Value := ;
*)



ExecuteSkill();

StepDone := ExecuteSkill.Done;
END_ACTION

ACTION ST42_CocktailOutput_active:
//RT: 2014.11.23: Ausgeben des Produktes
StepDone := FALSE;

//Skill auswählen
ExecuteSkill.SkillID 		:= 1403;
ExecuteSkill.SkillName	 	:= 'Output';

//Parameter setzen

ExecuteSkill.Parameter[1].ID := 1;
ExecuteSkill.Parameter[1].Name := 'TaskID';
ExecuteSkill.Parameter[1].Value := Order.TaskID;


(*
ExecuteSkill.Parameter[2].ID := ;
ExecuteSkill.Parameter[2].Name := '';
ExecuteSkill.Parameter[2].Value := ;
*)

(*
ExecuteSkill.Parameter[3].ID := ;
ExecuteSkill.Parameter[3].Name := '';
ExecuteSkill.Parameter[3].Value := ;
*)

(*
ExecuteSkill.Parameter[4].ID := ;
ExecuteSkill.Parameter[4].Name := '';
ExecuteSkill.Parameter[4].Value := ;
*)

(*
ExecuteSkill.Parameter[5].ID := ;
ExecuteSkill.Parameter[5].Name := '';
ExecuteSkill.Parameter[5].Value := ;
*)



ExecuteSkill();

StepDone := ExecuteSkill.Done;
END_ACTION

ACTION ST34_Exit_active:
SectionReady := TRUE;
END_ACTION

ACTION ST40_TransOutput_active:
//RT: 2014.11.23: Mover zum Output
StepDone := FALSE;

//Skill auswählen
ExecuteSkill.SkillID 		:= 1320;
ExecuteSkill.SkillName	 	:= 'Transport';

//Parameter setzen

ExecuteSkill.Parameter[3].ID := 3;
ExecuteSkill.Parameter[3].Name := 'Velocity';
ExecuteSkill.Parameter[3].Value := 300;



ExecuteSkill.Parameter[1].ID :=  1;
ExecuteSkill.Parameter[1].Name := 'TargetPosition X';
ExecuteSkill.Parameter[1].Value := 30 ;
ExecuteSkill.Parameter[1].StringValue := '#DP#2#XPosition';



ExecuteSkill.Parameter[2].ID := 2;
ExecuteSkill.Parameter[2].Name := 'TargetPosition Z';
ExecuteSkill.Parameter[2].Value := ZInputOutput;// ZCookieModule - ZCookieModuleCalibration - 2* Cookiethickness + toppingthickness+ Preasureheight  ;



(* ExecuteSkill.Parameter[4].ID := 4;
ExecuteSkill.Parameter[4].Name := 'Acceleration';
ExecuteSkill.Parameter[4].Value :=0 ;

*)
(*
ExecuteSkill.Parameter[5].ID := ;
ExecuteSkill.Parameter[5].Name := '';
ExecuteSkill.Parameter[5].Value := ;
*)



ExecuteSkill();

StepDone := ExecuteSkill.Done;
END_ACTION

ACTION ST33_UnblockPump_active:
//RT: 2014.11.23: Gibt Mover Position Frei
StepDone := FALSE;

//Skill auswählen
ExecuteSkill.SkillID 		:= 1316;
ExecuteSkill.SkillName	 	:= 'Unblock';

//Parameter setzen

ExecuteSkill.Parameter[1].ID := 1;
ExecuteSkill.Parameter[1].Name := 'TaskID';
ExecuteSkill.Parameter[1].Value := Order.TaskID;


(*
ExecuteSkill.Parameter[2].ID := ;
ExecuteSkill.Parameter[2].Name := '';
ExecuteSkill.Parameter[2].Value := ;
*)

(*
ExecuteSkill.Parameter[3].ID := ;
ExecuteSkill.Parameter[3].Name := '';
ExecuteSkill.Parameter[3].Value := ;
*)

(*
ExecuteSkill.Parameter[4].ID := ;
ExecuteSkill.Parameter[4].Name := '';
ExecuteSkill.Parameter[4].Value := ;
*)

(*
ExecuteSkill.Parameter[5].ID := ;
ExecuteSkill.Parameter[5].Name := '';
ExecuteSkill.Parameter[5].Value := ;
*)



ExecuteSkill();

StepDone := ExecuteSkill.Done;
END_ACTION

ACTION ST3_Pump_entry:
SectionReady := FALSE;
END_ACTION

ACTION ST4_Output_entry:
SectionReady := FALSE;
END_ACTION

ACTION ST5_Unreserve_active:
//RT: 2014.11.23: Mover Freigeben
StepDone := FALSE;

//Skill auswählen
ExecuteSkill.SkillID 		:= 1311;
ExecuteSkill.SkillName	 	:= 'Unreserve';

//Parameter setzen

ExecuteSkill.Parameter[1].ID := 1;
ExecuteSkill.Parameter[1].Name := 'TaskID';
ExecuteSkill.Parameter[1].Value := Order.TaskID;


(*
ExecuteSkill.Parameter[2].ID := ;
ExecuteSkill.Parameter[2].Name := '';
ExecuteSkill.Parameter[2].Val ue := ;
*)

(*
ExecuteSkill.Parameter[3].ID := ;
ExecuteSkill.Parameter[3].Name := '';
ExecuteSkill.Parameter[3].Value := ;
*)

(*
ExecuteSkill.Parameter[4].ID := ;
ExecuteSkill.Parameter[4].Name := '';
ExecuteSkill.Parameter[4].Value := ;
*)

(*
ExecuteSkill.Parameter[5].ID := ;
ExecuteSkill.Parameter[5].Name := '';
ExecuteSkill.Parameter[5].Value := ;
*)



ExecuteSkill();

StepDone := ExecuteSkill.Done;
END_ACTION

ACTION ST10_TransToInput_active:
//RT: 2014.11.23: Mover zum Input

StepDone := FALSE;

//Skill auswählen
ExecuteSkill.SkillID 		:= 1320;
ExecuteSkill.SkillName	 	:= 'Transport';

//Parameter setzen

ExecuteSkill.Parameter[3].ID := 3;
ExecuteSkill.Parameter[3].Name := 'Velocity';
ExecuteSkill.Parameter[3].Value := 1000;



ExecuteSkill.Parameter[1].ID :=  1;
ExecuteSkill.Parameter[1].Name := 'TargetPosition X';
ExecuteSkill.Parameter[1].Value := 30 ;
ExecuteSkill.Parameter[1].StringValue := '#DP#2#XPosition';



ExecuteSkill.Parameter[2].ID := 2;
ExecuteSkill.Parameter[2].Name := 'TargetPosition Z';
ExecuteSkill.Parameter[2].Value := 100;// ZCookieModule - ZCookieModuleCalibration - 2* Cookiethickness + toppingthickness+ Preasureheight  ;



(*
ExecuteSkill.Parameter[4].ID := 4;
ExecuteSkill.Parameter[4].Name := 'Acceleration';
ExecuteSkill.Parameter[4].Value := 0 ;
*)

(*
ExecuteSkill.Parameter[5].ID := ;
ExecuteSkill.Parameter[5].Name := '';
ExecuteSkill.Parameter[5].Value := ;
*)



ExecuteSkill();

StepDone := ExecuteSkill.Done;
END_ACTION

ACTION ST1_Input_entry:
SectionReady := FALSE;
END_ACTION

ACTION Init_active:
//RT: 2014.11.23: Vorbereiten der daten und der HMI
RecipeDone := FALSE;

// Initialisation of Recipe Parameters an name etc
RecipeInfo.Name := 'Pina Batida Lemon';
RecipeInfo.Description := 'Sour version of the classical Pina Colada Batida';
RecipeInfo.Dummy := FALSE;
RecipeInfo.RecipeID := 10059; 	// 
Initdone := TRUE;

//RT: 2014.11.23: wenn weniger als 5 alle lehren skills SkillID := 0
Command[1].SkillID := 1121;
Command[1].SkillName := 'Batida de Coco';
Command[1].Quantity := 35;

Command[2].SkillID := 1112;
Command[2].SkillName := 'Lemon Juice';
Command[2].Quantity := 10;

Command[3].SkillID := 1114;
Command[3].SkillName := 'Pineapple Juice';
Command[3].Quantity := 55;


Command[4].SkillID := 0;
Command[4].SkillName := 'Maracuja Juice';
Command[4].Quantity := 30;

Command[5].SkillID := 0;
Command[5].SkillName := 'Blue Curacao';
Command[5].Quantity := 10;








//Parameter 0:

	RecipeInfo.UserParameter[0].Dummy 		:= FALSE;
	RecipeInfo.UserParameter[0].Default		:= 200;
	RecipeInfo.UserParameter[0].Description	:= 'Gives the total fluid amount in the glass';
	RecipeInfo.UserParameter[0].MaxValue	:= 200;
	RecipeInfo.UserParameter[0].MinValue	:= 10;
	RecipeInfo.UserParameter[0].Name		:= 'Total Liquid Amount';
	RecipeInfo.UserParameter[0].Unit		:= 'ml';
	
//Parameter 1-5:
FOR i := 1 TO 5 DO
	IF Command[i].SkillID = 0 THEN
		RecipeInfo.UserParameter[i].Dummy 		:= TRUE;
	ELSE
		RecipeInfo.UserParameter[i].Dummy 		:= FALSE;
		RecipeInfo.UserParameter[i].Default		:= Command[i].Quantity;
		RecipeInfo.UserParameter[i].Description	:= Command[i].SkillName;
		RecipeInfo.UserParameter[i].MaxValue	:= 100;
		RecipeInfo.UserParameter[i].MinValue	:= 1;
		RecipeInfo.UserParameter[i].Name		:= Command[i].SkillName;
		RecipeInfo.UserParameter[i].Unit		:= 'ml';	
	END_IF
END_FOR
END_ACTION

ACTION ST0_Reserve_active:
//RT: 2014.11.23: Reservire einen Mover

StepDone := FALSE;
RecipeDone := FALSE;
//Skill auswählen
ExecuteSkill.SkillID 		:= 1310;
ExecuteSkill.SkillName	 	:= 'Reserve';

//Parameter setzen

ExecuteSkill.Parameter[1].ID := 1;
ExecuteSkill.Parameter[1].Name := 'TaskID';
ExecuteSkill.Parameter[1].Value := Order.TaskID;

(*
ExecuteSkill.Parameter[2].ID := ;
ExecuteSkill.Parameter[2].Name := '';
ExecuteSkill.Parameter[2].Value := ;
*)

(*
ExecuteSkill.Parameter[3].ID := ;
ExecuteSkill.Parameter[3].Name := '';
ExecuteSkill.Parameter[3].Value := ;
*)

(*
ExecuteSkill.Parameter[4].ID := ;
ExecuteSkill.Parameter[4].Name := '';
ExecuteSkill.Parameter[4].Value := ;
*)

(*
ExecuteSkill.Parameter[5].ID := ;
ExecuteSkill.Parameter[5].Name := '';
ExecuteSkill.Parameter[5].Value := ;
*)

ExecuteSkill();

StepDone := ExecuteSkill.Done;
END_ACTION

ACTION ST41_BlockOutput_active:
//RT: 2014.11.23: Blockirt den Mover an Position
StepDone := FALSE;

//Skill auswählen
ExecuteSkill.SkillID 		:= 1315;
ExecuteSkill.SkillName	 	:= 'Block';

//Parameter setzen

ExecuteSkill.Parameter[1].ID := 1;
ExecuteSkill.Parameter[1].Name := 'TaskID';
ExecuteSkill.Parameter[1].Value := Order.TaskID;


(*
ExecuteSkill.Parameter[2].ID := ;
ExecuteSkill.Parameter[2].Name := '';
ExecuteSkill.Parameter[2].Value := ;
*)

(*
ExecuteSkill.Parameter[3].ID := ;
ExecuteSkill.Parameter[3].Name := '';
ExecuteSkill.Parameter[3].Value := ;
*)

(*
ExecuteSkill.Parameter[4].ID := ;
ExecuteSkill.Parameter[4].Name := '';
ExecuteSkill.Parameter[4].Value := ;
*)

(*
ExecuteSkill.Parameter[5].ID := ;
ExecuteSkill.Parameter[5].Name := '';
ExecuteSkill.Parameter[5].Value := ;
*)



ExecuteSkill();

StepDone := ExecuteSkill.Done;
END_ACTION

ACTION ST30_TransPump_active:
//RT: 2014.11.23: Mover zum Pump
StepDone := FALSE;

//Skill auswählen
ExecuteSkill.SkillID 		:= 1320;
ExecuteSkill.SkillName	 	:= 'Transport';

//Parameter setzen

ExecuteSkill.Parameter[3].ID := 3;
ExecuteSkill.Parameter[3].Name := 'Velocity';
ExecuteSkill.Parameter[3].Value := 1000;



ExecuteSkill.Parameter[1].ID :=  1;
ExecuteSkill.Parameter[1].Name := 'TargetPosition X';
ExecuteSkill.Parameter[1].Value := 30 ;
ExecuteSkill.Parameter[1].StringValue := '#DP#2#XPosition';



ExecuteSkill.Parameter[2].ID := 2;
ExecuteSkill.Parameter[2].Name := 'TargetPosition Z';
ExecuteSkill.Parameter[2].Value := 25;// ZCookieModule - ZCookieModuleCalibration - 2* Cookiethickness + toppingthickness+ Preasureheight  ;



(*
ExecuteSkill.Parameter[4].ID := 4;
ExecuteSkill.Parameter[4].Name := 'Acceleration';
ExecuteSkill.Parameter[4].Value := 0 ;
*)

(*
ExecuteSkill.Parameter[5].ID := ;
ExecuteSkill.Parameter[5].Name := '';
ExecuteSkill.Parameter[5].Value := ;
*)



ExecuteSkill();

StepDone := ExecuteSkill.Done;
END_ACTION

ACTION ST1_Reserve0_active:
//RT: 2014.11.23: Reservire einen Mover

StepDone := FALSE;
RecipeDone := FALSE;
//Skill auswählen
ExecuteSkill.SkillID 		:= 1310;
ExecuteSkill.SkillName	 	:= 'Reserve';

//Parameter setzen

ExecuteSkill.Parameter[1].ID := 1;
ExecuteSkill.Parameter[1].Name := 'TaskID';
ExecuteSkill.Parameter[1].Value := Order.TaskID;

(*
ExecuteSkill.Parameter[2].ID := ;
ExecuteSkill.Parameter[2].Name := '';
ExecuteSkill.Parameter[2].Value := ;
*)

(*
ExecuteSkill.Parameter[3].ID := ;
ExecuteSkill.Parameter[3].Name := '';
ExecuteSkill.Parameter[3].Value := ;
*)

(*
ExecuteSkill.Parameter[4].ID := ;
ExecuteSkill.Parameter[4].Name := '';
ExecuteSkill.Parameter[4].Value := ;
*)

(*
ExecuteSkill.Parameter[5].ID := ;
ExecuteSkill.Parameter[5].Name := '';
ExecuteSkill.Parameter[5].Value := ;
*)

ExecuteSkill();

StepDone := ExecuteSkill.Done;
END_ACTION

ACTION ST1_Input_active:
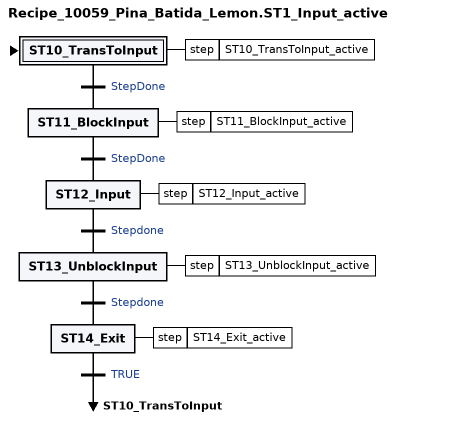
INITIAL_STEP ST10_TransToInput:
    ST10_TransToInput_active(N);  // step action
END_STEP
TRANSITION FROM ST10_TransToInput TO ST11_BlockInput
    := StepDone;
END_TRANSITION
STEP ST11_BlockInput:
    ST11_BlockInput_active(N);  // step action
END_STEP
TRANSITION FROM ST11_BlockInput TO ST12_Input
    := StepDone;
END_TRANSITION
STEP ST12_Input:
    ST12_Input_active(N);  // step action
END_STEP
TRANSITION FROM ST12_Input TO ST13_UnblockInput
    := Stepdone;
END_TRANSITION
STEP ST13_UnblockInput:
    ST13_UnblockInput_active(N);  // step action
END_STEP
TRANSITION FROM ST13_UnblockInput TO ST14_Exit
    := Stepdone;
END_TRANSITION
STEP ST14_Exit:
    ST14_Exit_active(N);  // step action
END_STEP
TRANSITION FROM ST14_Exit TO ST10_TransToInput
    := TRUE;
END_TRANSITION
END_ACTION

ACTION ST13_UnblockInput_active:
//RT: 2014.11.23: Gibt Mover Position Frei
StepDone := FALSE;

//Skill auswählen
ExecuteSkill.SkillID 		:= 1316;
ExecuteSkill.SkillName	 	:= 'Unblock';

//Parameter setzen

ExecuteSkill.Parameter[1].ID := 1;
ExecuteSkill.Parameter[1].Name := 'TaskID';
ExecuteSkill.Parameter[1].Value := Order.TaskID;


(*
ExecuteSkill.Parameter[2].ID := ;
ExecuteSkill.Parameter[2].Name := '';
ExecuteSkill.Parameter[2].Value := ;
*)

(*
ExecuteSkill.Parameter[3].ID := ;
ExecuteSkill.Parameter[3].Name := '';
ExecuteSkill.Parameter[3].Value := ;
*)

(*
ExecuteSkill.Parameter[4].ID := ;
ExecuteSkill.Parameter[4].Name := '';
ExecuteSkill.Parameter[4].Value := ;
*)

(*
ExecuteSkill.Parameter[5].ID := ;
ExecuteSkill.Parameter[5].Name := '';
ExecuteSkill.Parameter[5].Value := ;
*)



ExecuteSkill();

StepDone := ExecuteSkill.Done;
END_ACTION

ACTION ST14_Exit_active:
SectionReady := TRUE;
END_ACTION

ACTION ST4_Output_active:
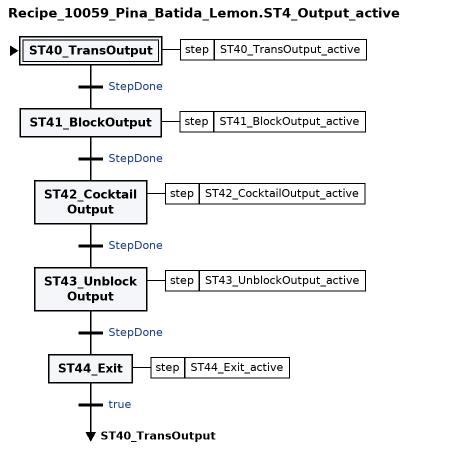
INITIAL_STEP ST40_TransOutput:
    ST40_TransOutput_active(N);  // step action
END_STEP
TRANSITION FROM ST40_TransOutput TO ST41_BlockOutput
    := StepDone;
END_TRANSITION
STEP ST41_BlockOutput:
    ST41_BlockOutput_active(N);  // step action
END_STEP
TRANSITION FROM ST41_BlockOutput TO ST42_CocktailOutput
    := StepDone;
END_TRANSITION
STEP ST42_CocktailOutput:
    ST42_CocktailOutput_active(N);  // step action
END_STEP
TRANSITION FROM ST42_CocktailOutput TO ST43_UnblockOutput
    := StepDone;
END_TRANSITION
STEP ST43_UnblockOutput:
    ST43_UnblockOutput_active(N);  // step action
END_STEP
TRANSITION FROM ST43_UnblockOutput TO ST44_Exit
    := StepDone;
END_TRANSITION
STEP ST44_Exit:
    ST44_Exit_active(N);  // step action
END_STEP
TRANSITION FROM ST44_Exit TO ST40_TransOutput
    := true;
END_TRANSITION
END_ACTION

ACTION ST3_Pump_active:
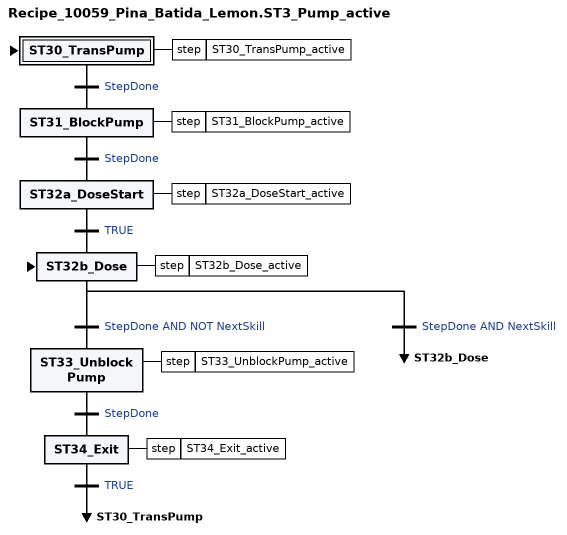
INITIAL_STEP ST30_TransPump:
    ST30_TransPump_active(N);  // step action
END_STEP
TRANSITION FROM ST30_TransPump TO ST31_BlockPump
    := StepDone;
END_TRANSITION
STEP ST31_BlockPump:
    ST31_BlockPump_active(N);  // step action
END_STEP
TRANSITION FROM ST31_BlockPump TO ST32a_DoseStart
    := StepDone;
END_TRANSITION
STEP ST32a_DoseStart:
    ST32a_DoseStart_active(N);  // step action
END_STEP
TRANSITION FROM ST32a_DoseStart TO ST32b_Dose
    := TRUE;
END_TRANSITION
STEP ST32b_Dose:
    ST32b_Dose_active(N);  // step action
END_STEP
TRANSITION FROM ST32b_Dose TO ST33_UnblockPump
    := StepDone AND NOT NextSkill;
END_TRANSITION
STEP ST33_UnblockPump:
    ST33_UnblockPump_active(N);  // step action
END_STEP
TRANSITION FROM ST33_UnblockPump TO ST34_Exit
    := StepDone;
END_TRANSITION
STEP ST34_Exit:
    ST34_Exit_active(N);  // step action
END_STEP
TRANSITION FROM ST34_Exit TO ST30_TransPump
    := TRUE;
END_TRANSITION
TRANSITION FROM ST32b_Dose TO ST32b_Dose
    := StepDone AND NextSkill;
END_TRANSITION
END_ACTION

ACTION ST44_Exit_active:
SectionReady := TRUE;
END_ACTION

ACTION ST43_UnblockOutput_active:
//RT: 2014.11.23: Gibt Mover Position Frei
StepDone := FALSE;

//Skill auswählen
ExecuteSkill.SkillID 		:= 1316;
ExecuteSkill.SkillName	 	:= 'Unblock';

//Parameter setzen

ExecuteSkill.Parameter[1].ID := 1;
ExecuteSkill.Parameter[1].Name := 'TaskID';
ExecuteSkill.Parameter[1].Value := Order.TaskID;


(*
ExecuteSkill.Parameter[2].ID := ;
ExecuteSkill.Parameter[2].Name := '';
ExecuteSkill.Parameter[2].Value := ;
*)

(*
ExecuteSkill.Parameter[3].ID := ;
ExecuteSkill.Parameter[3].Name := '';
ExecuteSkill.Parameter[3].Value := ;
*)

(*
ExecuteSkill.Parameter[4].ID := ;
ExecuteSkill.Parameter[4].Name := '';
ExecuteSkill.Parameter[4].Value := ;
*)

(*
ExecuteSkill.Parameter[5].ID := ;
ExecuteSkill.Parameter[5].Name := '';
ExecuteSkill.Parameter[5].Value := ;
*)



ExecuteSkill();

StepDone := ExecuteSkill.Done;
END_ACTION

ACTION ST31_BlockPump_active:
//RT: 2014.11.23: Blockirt den Mover an Position
StepDone := FALSE;

//Skill auswählen
ExecuteSkill.SkillID 		:= 1315;
ExecuteSkill.SkillName	 	:= 'Block';

//Parameter setzen

ExecuteSkill.Parameter[1].ID := 1;
ExecuteSkill.Parameter[1].Name := 'TaskID';
ExecuteSkill.Parameter[1].Value := Order.TaskID;


(*
ExecuteSkill.Parameter[2].ID := ;
ExecuteSkill.Parameter[2].Name := '';
ExecuteSkill.Parameter[2].Value := ;
*)

(*
ExecuteSkill.Parameter[3].ID := ;
ExecuteSkill.Parameter[3].Name := '';
ExecuteSkill.Parameter[3].Value := ;
*)

(*
ExecuteSkill.Parameter[4].ID := ;
ExecuteSkill.Parameter[4].Name := '';
ExecuteSkill.Parameter[4].Value := ;
*)

(*
ExecuteSkill.Parameter[5].ID := ;
ExecuteSkill.Parameter[5].Name := '';
ExecuteSkill.Parameter[5].Value := ;
*)



ExecuteSkill();

StepDone := ExecuteSkill.Done;
END_ACTION

ACTION ST32b_Dose_active:
//RT: 2014.11.23: Die Dosir Skills anlegen
StepDone := FALSE;

//Skill auswählen
ExecuteSkill.SkillID 		:= Command[i].SkillID;
ExecuteSkill.SkillName	 	:= Command[i].SkillName;
//Parameter setzen

ExecuteSkill.Parameter[0].ID := 1;
ExecuteSkill.Parameter[0].Name := 'Quantity';
//order.userParameter[0] = amount
ExecuteSkill.Parameter[0].Value := order.UserParameter[0].Value * order.UserParameter[i].Value / userparametersum ;//Summe aller Zutatenmengen;

(*
ExecuteSkill.Parameter[2].ID := ;
ExecuteSkill.Parameter[2].Name := '';
ExecuteSkill.Parameter[2].Value := ;
*)

(*
ExecuteSkill.Parameter[3].ID := ;
ExecuteSkill.Parameter[3].Name := '';
ExecuteSkill.Parameter[3].Value := ;
*)

(*
ExecuteSkill.Parameter[4].ID := ;
ExecuteSkill.Parameter[4].Name := '';
ExecuteSkill.Parameter[4].Value := ;
*)

(*
ExecuteSkill.Parameter[5].ID := ;
ExecuteSkill.Parameter[5].Name := '';
ExecuteSkill.Parameter[5].Value := ;
*)


ExecuteSkill();

StepDone := ExecuteSkill.Done;

i := i + 1 ;

IF i = 6 THEN
	NextSkill := FALSE;
ELSIF Command[i].SkillID = 0 THEN
	NextSkill := FALSE;
ELSE
	NextSkill := TRUE;
END_IF
END_ACTION

END_FUNCTION_BLOCK

// ---- POUs/Recipes/Recipe_10058_RedOne.TcPOU
FUNCTION_BLOCK Recipe_10058_RedOne
VAR_INPUT
	execute: BOOL;
	Order: DUT_RECIPEORDER;
END_VAR
VAR_OUTPUT
	RecipeInfo: DUT_RECIPEOFFER;
	RecipeDone: BOOL;
	InitDone: BOOL;
	Ready: BOOL;
END_VAR
VAR
	userparametersum: LREAL;
	StepDone: BOOL;
	i: INT;
	Command: ARRAY[1..5] OF DUT_RecipeCommand;
	NextSkill: BOOL;
	SectionReady: BOOL;
END_VAR

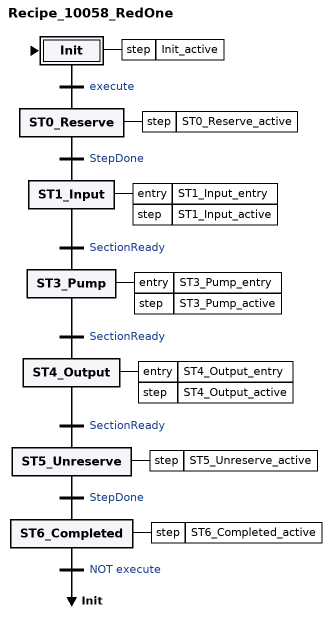
INITIAL_STEP Init:
    Init_active(N);  // step action
END_STEP
TRANSITION FROM Init TO ST0_Reserve
    := execute;
END_TRANSITION
STEP ST0_Reserve:
    ST0_Reserve_active(N);  // step action
END_STEP
TRANSITION FROM ST0_Reserve TO ST1_Input
    := StepDone;
END_TRANSITION
STEP ST1_Input:
    ST1_Input_entry(P1);  // entry action
    ST1_Input_active(N);  // step action
END_STEP
TRANSITION FROM ST1_Input TO ST3_Pump
    := SectionReady;
END_TRANSITION
STEP ST3_Pump:
    ST3_Pump_entry(P1);  // entry action
    ST3_Pump_active(N);  // step action
END_STEP
TRANSITION FROM ST3_Pump TO ST4_Output
    := SectionReady;
END_TRANSITION
STEP ST4_Output:
    ST4_Output_entry(P1);  // entry action
    ST4_Output_active(N);  // step action
END_STEP
TRANSITION FROM ST4_Output TO ST5_Unreserve
    := SectionReady;
END_TRANSITION
STEP ST5_Unreserve:
    ST5_Unreserve_active(N);  // step action
END_STEP
TRANSITION FROM ST5_Unreserve TO ST6_Completed
    := StepDone;
END_TRANSITION
STEP ST6_Completed:
    ST6_Completed_active(N);  // step action
END_STEP
TRANSITION FROM ST6_Completed TO Init
    := NOT execute;
END_TRANSITION

ACTION ST14_Exit_active:
SectionReady := TRUE;
END_ACTION

ACTION ST12_Input_active:
//RT: 2014.11.23: Input Modul auslösen
StepDone := FALSE;

//Skill auswählen
ExecuteSkill.SkillID 		:= 1402;
ExecuteSkill.SkillName	 	:= 'Input';

//Parameter setzen

ExecuteSkill.Parameter[1].ID := 1;
ExecuteSkill.Parameter[1].Name := 'TaskID';
ExecuteSkill.Parameter[1].Value := Order.TaskID;


(*
ExecuteSkill.Parameter[2].ID := ;
ExecuteSkill.Parameter[2].Name := '';
ExecuteSkill.Parameter[2].Value := ;
*)

(*
ExecuteSkill.Parameter[3].ID := ;
ExecuteSkill.Parameter[3].Name := '';
ExecuteSkill.Parameter[3].Value := ;
*)

(*
ExecuteSkill.Parameter[4].ID := ;
ExecuteSkill.Parameter[4].Name := '';
ExecuteSkill.Parameter[4].Value := ;
*)

(*
ExecuteSkill.Parameter[5].ID := ;
ExecuteSkill.Parameter[5].Name := '';
ExecuteSkill.Parameter[5].Value := ;
*)



ExecuteSkill();

StepDone := ExecuteSkill.Done;
END_ACTION

ACTION ST34_Exit_active:
SectionReady := TRUE;
END_ACTION

ACTION ST41_BlockOutput_active:
//RT: 2014.11.23: Blockirt den Mover an Position
StepDone := FALSE;

//Skill auswählen
ExecuteSkill.SkillID 		:= 1315;
ExecuteSkill.SkillName	 	:= 'Block';

//Parameter setzen

ExecuteSkill.Parameter[1].ID := 1;
ExecuteSkill.Parameter[1].Name := 'TaskID';
ExecuteSkill.Parameter[1].Value := Order.TaskID;


(*
ExecuteSkill.Parameter[2].ID := ;
ExecuteSkill.Parameter[2].Name := '';
ExecuteSkill.Parameter[2].Value := ;
*)

(*
ExecuteSkill.Parameter[3].ID := ;
ExecuteSkill.Parameter[3].Name := '';
ExecuteSkill.Parameter[3].Value := ;
*)

(*
ExecuteSkill.Parameter[4].ID := ;
ExecuteSkill.Parameter[4].Name := '';
ExecuteSkill.Parameter[4].Value := ;
*)

(*
ExecuteSkill.Parameter[5].ID := ;
ExecuteSkill.Parameter[5].Name := '';
ExecuteSkill.Parameter[5].Value := ;
*)



ExecuteSkill();

StepDone := ExecuteSkill.Done;
END_ACTION

ACTION ST13_UnblockInput_active:
//RT: 2014.11.23: Gibt Mover Position Frei
StepDone := FALSE;

//Skill auswählen
ExecuteSkill.SkillID 		:= 1316;
ExecuteSkill.SkillName	 	:= 'Unblock';

//Parameter setzen

ExecuteSkill.Parameter[1].ID := 1;
ExecuteSkill.Parameter[1].Name := 'TaskID';
ExecuteSkill.Parameter[1].Value := Order.TaskID;


(*
ExecuteSkill.Parameter[2].ID := ;
ExecuteSkill.Parameter[2].Name := '';
ExecuteSkill.Parameter[2].Value := ;
*)

(*
ExecuteSkill.Parameter[3].ID := ;
ExecuteSkill.Parameter[3].Name := '';
ExecuteSkill.Parameter[3].Value := ;
*)

(*
ExecuteSkill.Parameter[4].ID := ;
ExecuteSkill.Parameter[4].Name := '';
ExecuteSkill.Parameter[4].Value := ;
*)

(*
ExecuteSkill.Parameter[5].ID := ;
ExecuteSkill.Parameter[5].Name := '';
ExecuteSkill.Parameter[5].Value := ;
*)



ExecuteSkill();

StepDone := ExecuteSkill.Done;
END_ACTION

ACTION ST4_Output_active:
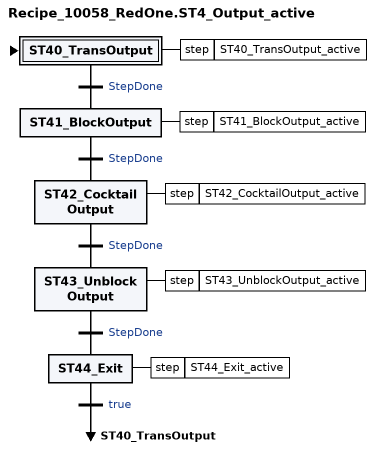
INITIAL_STEP ST40_TransOutput:
    ST40_TransOutput_active(N);  // step action
END_STEP
TRANSITION FROM ST40_TransOutput TO ST41_BlockOutput
    := StepDone;
END_TRANSITION
STEP ST41_BlockOutput:
    ST41_BlockOutput_active(N);  // step action
END_STEP
TRANSITION FROM ST41_BlockOutput TO ST42_CocktailOutput
    := StepDone;
END_TRANSITION
STEP ST42_CocktailOutput:
    ST42_CocktailOutput_active(N);  // step action
END_STEP
TRANSITION FROM ST42_CocktailOutput TO ST43_UnblockOutput
    := StepDone;
END_TRANSITION
STEP ST43_UnblockOutput:
    ST43_UnblockOutput_active(N);  // step action
END_STEP
TRANSITION FROM ST43_UnblockOutput TO ST44_Exit
    := StepDone;
END_TRANSITION
STEP ST44_Exit:
    ST44_Exit_active(N);  // step action
END_STEP
TRANSITION FROM ST44_Exit TO ST40_TransOutput
    := true;
END_TRANSITION
END_ACTION

ACTION ST42_CocktailOutput_active:
//RT: 2014.11.23: Ausgeben des Produktes
StepDone := FALSE;

//Skill auswählen
ExecuteSkill.SkillID 		:= 1403;
ExecuteSkill.SkillName	 	:= 'Output';

//Parameter setzen

ExecuteSkill.Parameter[1].ID := 1;
ExecuteSkill.Parameter[1].Name := 'TaskID';
ExecuteSkill.Parameter[1].Value := Order.TaskID;


(*
ExecuteSkill.Parameter[2].ID := ;
ExecuteSkill.Parameter[2].Name := '';
ExecuteSkill.Parameter[2].Value := ;
*)

(*
ExecuteSkill.Parameter[3].ID := ;
ExecuteSkill.Parameter[3].Name := '';
ExecuteSkill.Parameter[3].Value := ;
*)

(*
ExecuteSkill.Parameter[4].ID := ;
ExecuteSkill.Parameter[4].Name := '';
ExecuteSkill.Parameter[4].Value := ;
*)

(*
ExecuteSkill.Parameter[5].ID := ;
ExecuteSkill.Parameter[5].Name := '';
ExecuteSkill.Parameter[5].Value := ;
*)



ExecuteSkill();

StepDone := ExecuteSkill.Done;
END_ACTION

ACTION ST40_TransOutput_active:
//RT: 2014.11.23: Mover zum Output
StepDone := FALSE;

//Skill auswählen
ExecuteSkill.SkillID 		:= 1320;
ExecuteSkill.SkillName	 	:= 'Transport';

//Parameter setzen

ExecuteSkill.Parameter[3].ID := 3;
ExecuteSkill.Parameter[3].Name := 'Velocity';
ExecuteSkill.Parameter[3].Value := 300;



ExecuteSkill.Parameter[1].ID :=  1;
ExecuteSkill.Parameter[1].Name := 'TargetPosition X';
ExecuteSkill.Parameter[1].Value := 30 ;
ExecuteSkill.Parameter[1].StringValue := '#DP#2#XPosition';



ExecuteSkill.Parameter[2].ID := 2;
ExecuteSkill.Parameter[2].Name := 'TargetPosition Z';
ExecuteSkill.Parameter[2].Value := 100;// ZCookieModule - ZCookieModuleCalibration - 2* Cookiethickness + toppingthickness+ Preasureheight  ;



(* ExecuteSkill.Parameter[4].ID := 4;
ExecuteSkill.Parameter[4].Name := 'Acceleration';
ExecuteSkill.Parameter[4].Value :=0 ;

*)
(*
ExecuteSkill.Parameter[5].ID := ;
ExecuteSkill.Parameter[5].Name := '';
ExecuteSkill.Parameter[5].Value := ;
*)



ExecuteSkill();

StepDone := ExecuteSkill.Done;
END_ACTION

